{attribute 'TcRpcEnable' := '1'}
METHOD CheckState : HRESULT
VAR_INPUT
	hdl : UDINT; // Do not change, used by server.
END_VAR
VAR_OUTPUT
	bBusy : BOOL; // Do not change. Used by server to find out if the job is finished
	
	// List of OutputArguments for OPC UA method, may be customized
	State : BOOL; // Abgeschlossener MethodCall
	MethodCall: BOOL; //Input Recall
END_VAR
                        callCounterCheckState := callCounterCheckState + 1;
IF NOT jobFinished THEN
	bBusy := TRUE; // job is not finished yet
	CheckState := 0; // no error
ELSE
	bBusy := FALSE; // job is finished
	CheckState := 0; // done, no error occured during execution (OPC UA StatusCode "GOOD")
	jobFinished := FALSE;
	State := ResetCall;
	MethodCall := MethodCall_Name;
END_IF
                      
END_METHOD

{attribute 'TcRpcEnable' := '1'}
METHOD Start : HRESULT
VAR_INPUT
	// List of InputArguments for OPC UA method, may be customized
	MethodCall : BOOL; // some description
	DirectionPointA : BOOL;
	DirectionPointB : BOOL;
	EndschalterEntlastung : BOOL;	
END_VAR
VAR_OUTPUT
	hdl : UDINT; // Do not change, used by server.
END_VAR
                        callCounterStart := callCounterStart + 1;

MethodCall_Name := MethodCall;
DirectionPointA := Direction_01;
DirectionPointB := Direction_02;
EndschalterEntlastung := EndschalterEntlastung;

IF DirectionPointA := TRUE THEN
	DirectionPointB := FALSE;
END_IF

IF DirectionPointB := TRUE THEN
	DirectionPointA := FALSE;
END_IF

jobRunning := TRUE;
Start := 0; // no error occured, e.g. while parsing the input arguments (0 = OPC UA StatusCode "GOOD")
                      
END_METHOD
END_FUNCTION_BLOCK

FUNCTION_BLOCK HRL_OperatingModes
VAR_INPUT
	Start 			: BOOL;
	Stop			: BOOL;
	Reset			: BOOL;
	Schalter		: BOOL;
	Schrittkette_GS	: BOOL;
	Count1 : INT := 0;
	Count2 : INT := 0;
	Alt_abort: BOOL;
	Err_detected: BOOL;
	Diag_finished: BOOL;
	Alt_found: BOOL;
	Cycle_finished: BOOL;

END_VAR
VAR_OUTPUT
	{attribute 'OPC.UA.DA' := '1'} // für OPC UA freigeben
	A1 : BOOL := FALSE; //Initialzustand
	{attribute 'OPC.UA.DA' := '1'} // für OPC UA freigeben
	A2 : BOOL; //Stillstand angefordert am Ende des Zyklus
//	A3 : BOOL; //Stillstand angefordert in einem bestimmten Zustand
//	A4 : BOOL; //Erhaltener Stillstand
	{attribute 'OPC.UA.DA' := '1'} // für OPC UA freigeben
	A5 : BOOL; //Vorbereitung zur Wiederaufnahme nach Störung
	{attribute 'OPC.UA.DA' := '1'} // für OPC UA freigeben
	A6 : BOOL; //Fahrt in den Initialzustand
	{attribute 'OPC.UA.DA' := '1'} // für OPC UA freigeben
	F1 : BOOL; //Normalbetrieb
//	F2 : BOOL; //Anfahren
//	F3 : BOOL; //Abfahren
	{attribute 'OPC.UA.DA' := '1'} // für OPC UA freigeben
	F4 : BOOL; //Handbetrieb
//	F5 : BOOL; //Schrittbetrieb
//	F6 : BOOL; //Testbetrieb
	{attribute 'OPC.UA.DA' := '1'} // für OPC UA freigeben
	D1 : BOOL; //Not-Aus
	{attribute 'OPC.UA.DA' := '1'} // für OPC UA freigeben
	D2 : BOOL; //Diagnose und Störbehandlung
	{attribute 'OPC.UA.DA' := '1'} // für OPC UA freigeben
	D3 : BOOL; //Produktion trotz Störung
	MethodCall_InitStateDrive : BOOL;
	InputVar_InitStateDrive : BOOL;
END_VAR
VAR
	bFirstScan : BOOL := TRUE;
	FirstScanCount: INT := 0;
	AlwaysTrue : BOOL := TRUE;
	TestingVariable : BOOL;	
	 nTaskIdx : DINT;
	RS_InitialState: RS;
	RS_InitialState11: RS;	
	RS_InitialDrive: RS;
	RS_ManualOperationMode: RS;
	RS_AutomaticOperationMode: RS;
	RS_CycleEnded: RS;
	//Count: INT := 0;
	R_TRIG_Manual: R_TRIG;
	R_TRIG_Automatic: R_TRIG;
	R_TRIG_InitialDrive: R_TRIG;
	R_TRIG_CycleEnded: R_TRIG;
	R_TRIG_Init: R_TRIG;
	NeverTrue: BOOL := FALSE;
	SR_D1: SR;
	RS_D2: RS;
	
	RS_D3: RS;
	RS_A5: RS;
	
	
	bFirstCycle: BOOL;
END_VAR
  VAR  (* added by the conversion: wires and edge detectors of the diagram *)
    _EXECUTE50000000009_EN : BOOL;
  END_VAR

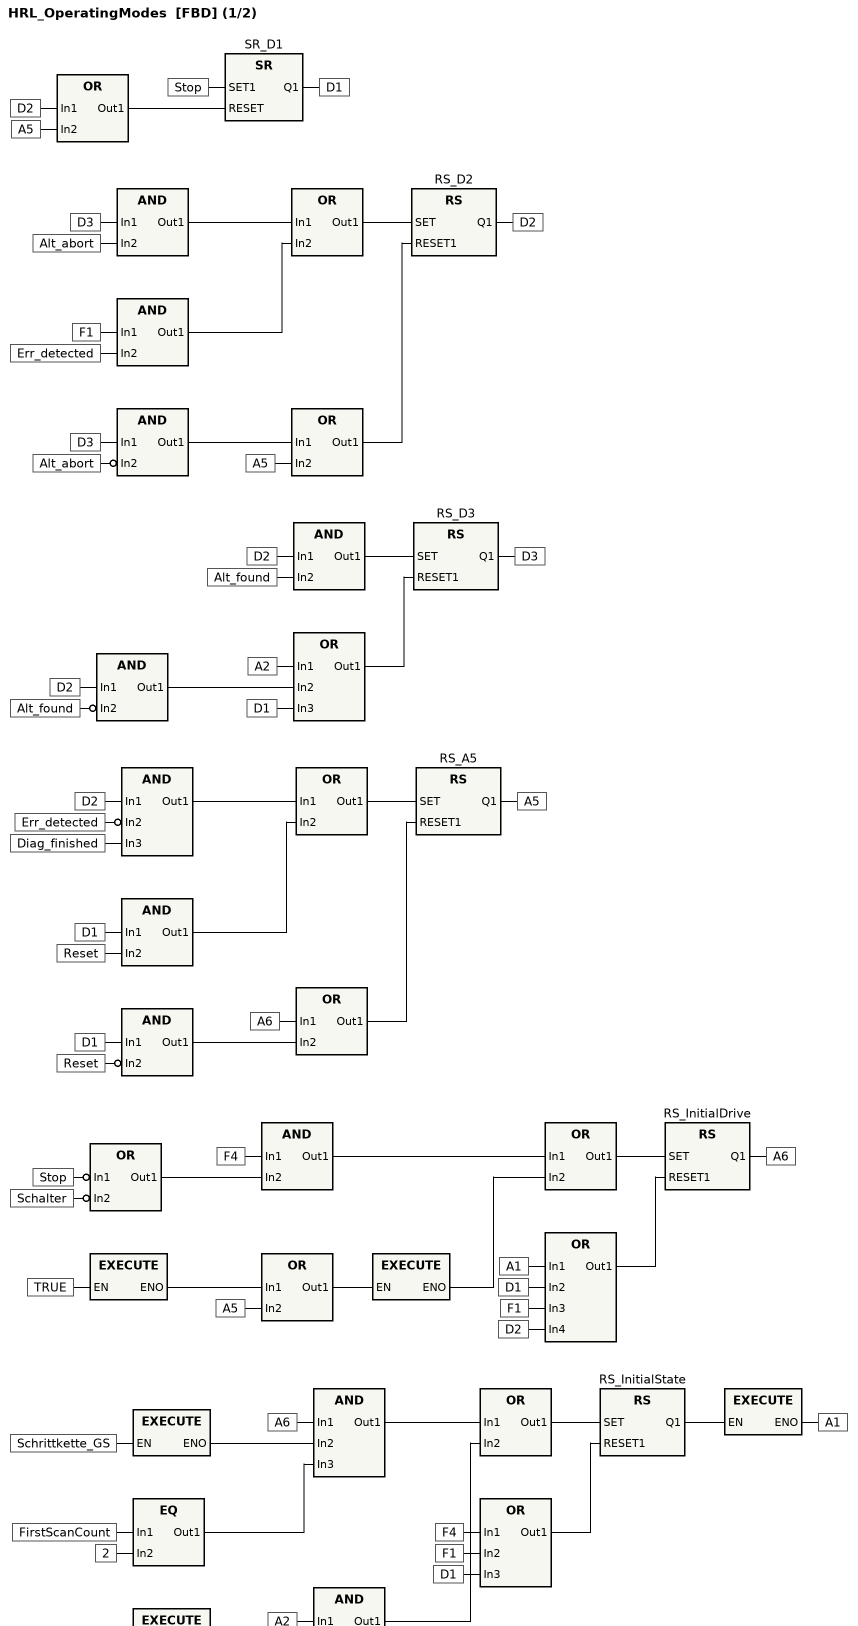
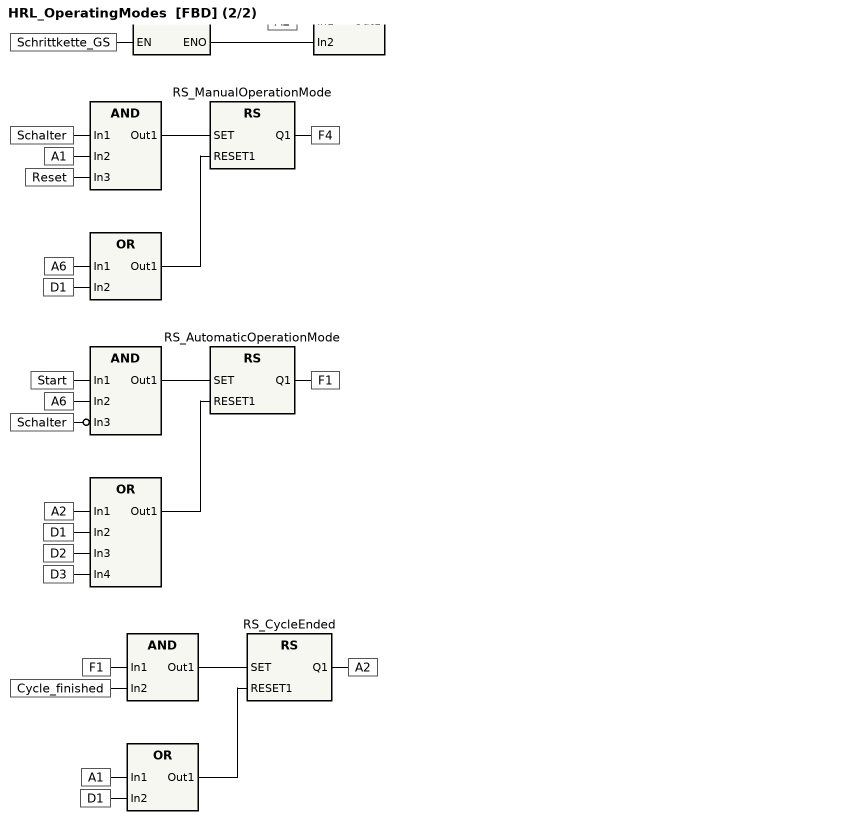
(* FBD diagram, written out as Structured Text *)
SR_D1(SET1 := Stop, RESET := D2 OR A5);
D1 := SR_D1.Q1;
RS_D2(SET := D3 AND Alt_abort OR F1 AND Err_detected, RESET1 := D3 AND NOT Alt_abort OR A5);
D2 := RS_D2.Q1;
RS_D3(SET := D2 AND Alt_found, RESET1 := A2 OR D2 AND NOT Alt_found OR D1);
D3 := RS_D3.Q1;
RS_A5(SET := D2 AND NOT Err_detected AND Diag_finished OR D1 AND Reset, RESET1 := A6 OR D1 AND NOT Reset);
A5 := RS_A5.Q1;
IF TRUE THEN
  nTaskIdx := GETCURTASKINDEXEX();
  
  IF nTaskIdx > 0 THEN
          bFirstCycle := _TaskInfo[nTaskIdx].FirstCycle;
  END_IF
END_IF;
_EXECUTE50000000009_EN := TRUE OR A5;
IF _EXECUTE50000000009_EN THEN
  IF AlwaysTrue THEN
      MethodCall_InitStateDrive := TRUE;
  	InputVar_InitStateDrive := TRUE;
  END_IF;
END_IF;
RS_InitialDrive(SET := F4 AND (NOT Stop OR NOT Schalter) OR _EXECUTE50000000009_EN, RESET1 := A1 OR D1 OR F1 OR D2);
A6 := RS_InitialDrive.Q1;
IF Schrittkette_GS THEN
  MethodCall_InitStateDrive := FALSE;
  InputVar_InitStateDrive := FALSE;
END_IF;
IF Schrittkette_GS THEN
  MethodCall_InitStateDrive := FALSE;
  InputVar_InitStateDrive := FALSE;
END_IF;
RS_InitialState(SET := A6 AND Schrittkette_GS AND FirstScanCount = 2 OR A2 AND Schrittkette_GS, RESET1 := F4 OR F1 OR D1);
IF RS_InitialState.Q1 THEN
  FirstScanCount := 0;
  bFirstScan := FALSE;
END_IF;
A1 := RS_InitialState.Q1;
RS_ManualOperationMode(SET := Schalter AND A1 AND Reset, RESET1 := A6 OR D1);
F4 := RS_ManualOperationMode.Q1;
RS_AutomaticOperationMode(SET := Start AND A6 AND NOT Schalter, RESET1 := A2 OR D1 OR D2 OR D3);
F1 := RS_AutomaticOperationMode.Q1;
RS_CycleEnded(SET := F1 AND Cycle_finished, RESET1 := A1 OR D1);
A2 := RS_CycleEnded.Q1;
END_FUNCTION_BLOCK

FUNCTION_BLOCK VSG_OperatingModes
VAR_INPUT
	Start 			: BOOL;
	Stop			: BOOL;
	Reset			: BOOL;
	Schalter		: BOOL;
	Schrittkette_GS	: BOOL;
	Count1 : INT := 0;
	Count2 : INT := 0;
	Alt_abort: BOOL;
	Err_detected: BOOL;
	Diag_finished: BOOL;
	Alt_found: BOOL;
	Cycle_finished: BOOL;

END_VAR
VAR_OUTPUT
	{attribute 'OPC.UA.DA' := '1'} // für OPC UA freigeben
	A1 : BOOL := FALSE; //Initialzustand
	{attribute 'OPC.UA.DA' := '1'} // für OPC UA freigeben
	A2 : BOOL; //Stillstand angefordert am Ende des Zyklus
//	A3 : BOOL; //Stillstand angefordert in einem bestimmten Zustand
//	A4 : BOOL; //Erhaltener Stillstand
	{attribute 'OPC.UA.DA' := '1'} // für OPC UA freigeben
	A5 : BOOL; //Vorbereitung zur Wiederaufnahme nach Störung
	{attribute 'OPC.UA.DA' := '1'} // für OPC UA freigeben
	A6 : BOOL; //Fahrt in den Initialzustand
	{attribute 'OPC.UA.DA' := '1'} // für OPC UA freigeben
	F1 : BOOL; //Normalbetrieb
//	F2 : BOOL; //Anfahren
//	F3 : BOOL; //Abfahren
	{attribute 'OPC.UA.DA' := '1'} // für OPC UA freigeben
	F4 : BOOL; //Handbetrieb
//	F5 : BOOL; //Schrittbetrieb
//	F6 : BOOL; //Testbetrieb
{attribute 'OPC.UA.DA' := '1'} // für OPC UA freigeben
	D1 : BOOL; //Not-Aus
	{attribute 'OPC.UA.DA' := '1'} // für OPC UA freigeben
	D2 : BOOL; //Diagnose und Störbehandlung
	{attribute 'OPC.UA.DA' := '1'} // für OPC UA freigeben
	D3 : BOOL; //Produktion trotz Störung
	MethodCall_InitStateDrive : BOOL;
	InputVar_InitStateDrive : BOOL;
END_VAR
VAR
	bFirstScan : BOOL := TRUE;
	FirstScanCount: INT := 0;
	AlwaysTrue : BOOL := TRUE;
	TestingVariable : BOOL;	
	 nTaskIdx : DINT;
	RS_InitialState: RS;
	RS_InitialState11: RS;	
	RS_InitialDrive: RS;
	RS_ManualOperationMode: RS;
	RS_AutomaticOperationMode: RS;
	RS_CycleEnded: RS;
	//Count: INT := 0;
	R_TRIG_Manual: R_TRIG;
	R_TRIG_Automatic: R_TRIG;
	R_TRIG_InitialDrive: R_TRIG;
	R_TRIG_CycleEnded: R_TRIG;
	R_TRIG_Init: R_TRIG;
	NeverTrue: BOOL := FALSE;
	SR_D1: SR;
	RS_D2: RS;
	
	RS_D3: RS;
	RS_A5: RS;
	
	
	bFirstCycle: BOOL;
END_VAR
  VAR  (* added by the conversion: wires and edge detectors of the diagram *)
    _EXECUTE50000000009_EN : BOOL;
  END_VAR

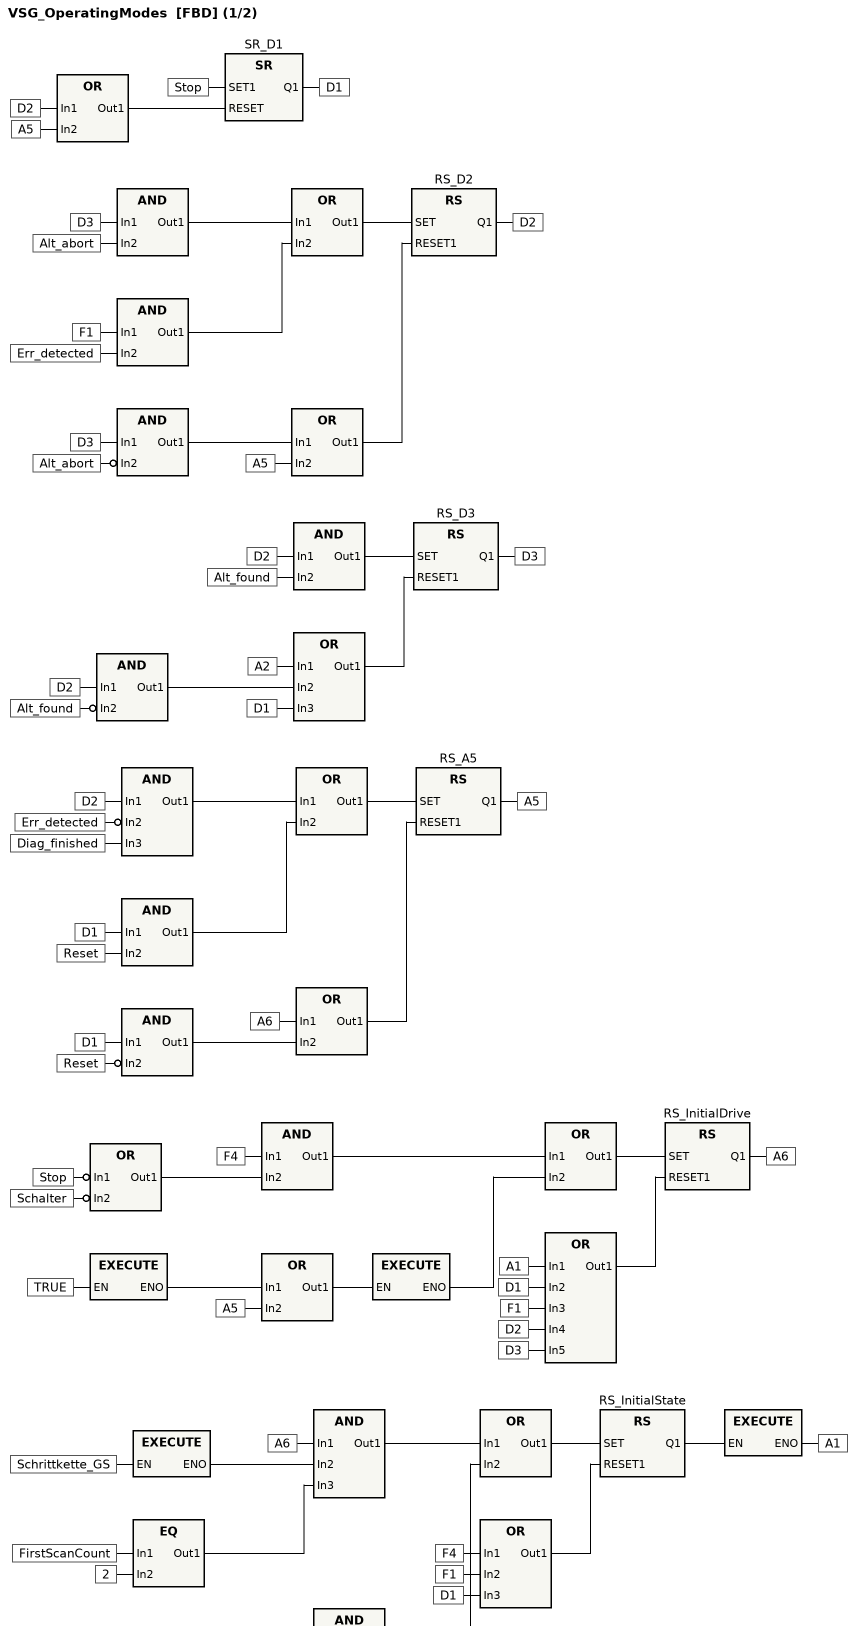
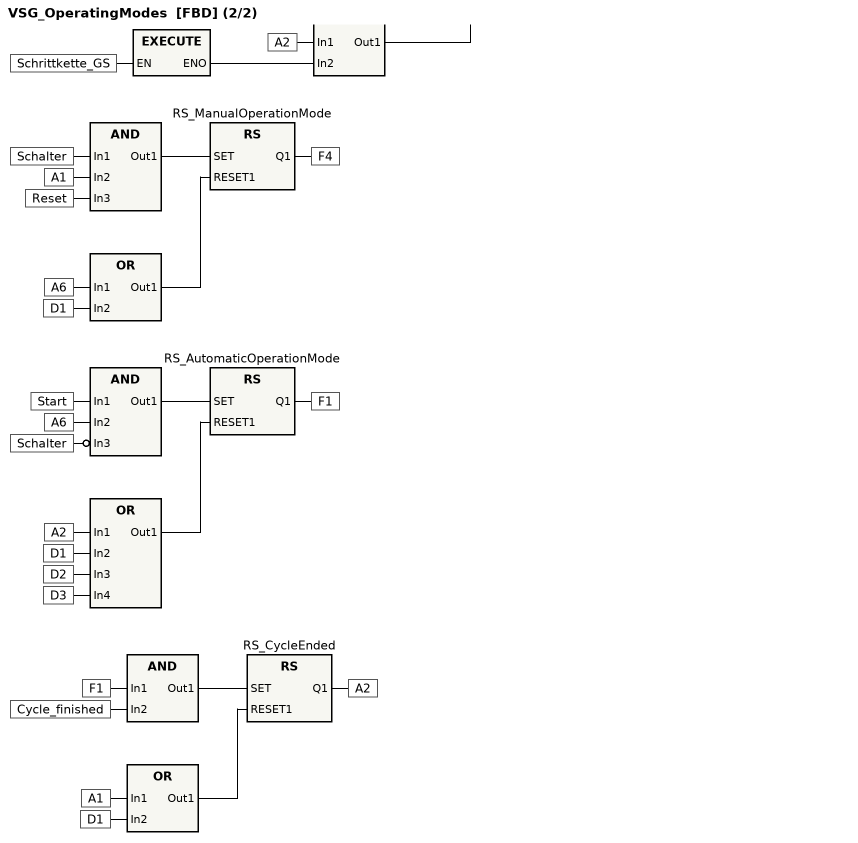
(* FBD diagram, written out as Structured Text *)
SR_D1(SET1 := Stop, RESET := D2 OR A5);
D1 := SR_D1.Q1;
RS_D2(SET := D3 AND Alt_abort OR F1 AND Err_detected, RESET1 := D3 AND NOT Alt_abort OR A5);
D2 := RS_D2.Q1;
RS_D3(SET := D2 AND Alt_found, RESET1 := A2 OR D2 AND NOT Alt_found OR D1);
D3 := RS_D3.Q1;
RS_A5(SET := D2 AND NOT Err_detected AND Diag_finished OR D1 AND Reset, RESET1 := A6 OR D1 AND NOT Reset);
A5 := RS_A5.Q1;
IF TRUE THEN
  nTaskIdx := GETCURTASKINDEXEX();
  
  IF nTaskIdx > 0 THEN
          bFirstCycle := _TaskInfo[nTaskIdx].FirstCycle;
  END_IF
END_IF;
_EXECUTE50000000009_EN := TRUE OR A5;
IF _EXECUTE50000000009_EN THEN
  IF AlwaysTrue THEN
      MethodCall_InitStateDrive := TRUE;
  	InputVar_InitStateDrive := TRUE;
  END_IF;
END_IF;
RS_InitialDrive(SET := F4 AND (NOT Stop OR NOT Schalter) OR _EXECUTE50000000009_EN, RESET1 := A1 OR D1 OR F1 OR D2 OR D3);
A6 := RS_InitialDrive.Q1;
IF Schrittkette_GS THEN
  MethodCall_InitStateDrive := FALSE;
  InputVar_InitStateDrive := FALSE;
END_IF;
IF Schrittkette_GS THEN
  MethodCall_InitStateDrive := FALSE;
  InputVar_InitStateDrive := FALSE;
END_IF;
RS_InitialState(SET := A6 AND Schrittkette_GS AND FirstScanCount = 2 OR A2 AND Schrittkette_GS, RESET1 := F4 OR F1 OR D1);
IF RS_InitialState.Q1 THEN
  FirstScanCount := 0;
  bFirstScan := FALSE;
END_IF;
A1 := RS_InitialState.Q1;
RS_ManualOperationMode(SET := Schalter AND A1 AND Reset, RESET1 := A6 OR D1);
F4 := RS_ManualOperationMode.Q1;
RS_AutomaticOperationMode(SET := Start AND A6 AND NOT Schalter, RESET1 := A2 OR D1 OR D2 OR D3);
F1 := RS_AutomaticOperationMode.Q1;
RS_CycleEnded(SET := F1 AND Cycle_finished, RESET1 := A1 OR D1);
A2 := RS_CycleEnded.Q1;
END_FUNCTION_BLOCK

FUNCTION_BLOCK MBS_OperatingModes
VAR_INPUT
	Start 			: BOOL;
	Stop			: BOOL;
	Reset			: BOOL;
	Schalter		: BOOL;
	Schrittkette_GS : BOOL;
END_VAR
VAR_OUTPUT
	A1 : BOOL; //Initialzustand
	A2 : BOOL; //Stillstand angefordert am Ende des Zyklus
//	A3 : BOOL; //Stillstand angefordert in einem bestimmten Zustand
//	A4 : BOOL; //Erhaltener Stillstand
//	A5 : BOOL; //Vorbereitung zur Wiederaufnahme nach Störung
	A6 : BOOL; //Fahrt in den Initialzustand
	F1 : BOOL; //Normalbetrieb
//	F2 : BOOL; //Anfahren
//	F3 : BOOL; //Abfahren
	F4 : BOOL; //Handbetrieb
//	F5 : BOOL; //Schrittbetrieb
//	F6 : BOOL; //Testbetrieb
//	D1 : BOOL; //Not-Aus
//	D2 : BOOL; //DIagnose und Störbehandlung
//	D3 : BOOL; //Produktion trotz Störung
END_VAR
VAR
	bFirstScan : BOOL := TRUE;	
	
	RS_InitialState: RS;	
	RS_InitialDrive: RS;
	RS_ManualOperationMode: RS;
	RS_AutomaticOperationMode: RS;
	RS_CycleEnded: RS;

	R_TRIG_Manual: R_TRIG;
	R_TRIG_Automatic: R_TRIG;
	R_TRIG_InitialDrive: R_TRIG;
	R_TRIG_CycleEnded: R_TRIG;
	R_TRIG_Init: R_TRIG;
END_VAR

                  R_TRIG_InitialDrive(CLK := RS_InitialDrive);
R_TRIG_CycleEnded(CLK := RS_CycleEnded);
R_TRIG_Manual(CLK := RS_ManualOperationMode);
R_TRIG_Automatic(CLK := RS_AutomaticOperationMode);
RS_InitialState(SET := ((((R_TRIG_InitialDrive.Q) AND (Schrittkette_GS))) OR (((R_TRIG_CycleEnded.Q) AND (Schrittkette_GS)))), RESET1 := ((R_TRIG_Manual.Q) OR (R_TRIG_Automatic.Q)));
A1 := RS_InitialState.Q1;
RS_ManualOperationMode(SET := ((Schalter) AND (A1) AND (Reset)), RESET1 := A6);
F4 := RS_ManualOperationMode.Q1;
R_TRIG_Manual(CLK := RS_ManualOperationMode);
R_TRIG_Init(CLK := RS_InitialState);
RS_InitialDrive(SET := ((((R_TRIG_Manual.Q) AND (((Stop) OR (NOT (Schalter)))))) OR ((bFirstScan))), RESET1 := R_TRIG_Init.Q);
A6 := RS_InitialDrive.Q1;
R_TRIG_Init(CLK := RS_InitialState);
R_TRIG_CycleEnded(CLK := RS_CycleEnded);
RS_AutomaticOperationMode(SET := ((Start) AND (R_TRIG_Init.Q) AND (NOT (Schalter))), RESET1 := R_TRIG_CycleEnded.Q);
F1 := RS_AutomaticOperationMode.Q1;
R_TRIG_Automatic(CLK := RS_AutomaticOperationMode);
R_TRIG_Init(CLK := RS_InitialState);
RS_CycleEnded(SET := ((R_TRIG_Automatic.Q) AND (((Schalter) OR (Stop)))), RESET1 := R_TRIG_Init.Q);
A2 := RS_CycleEnded.Q1;
                
END_FUNCTION_BLOCK

FUNCTION_BLOCK SST_OperatingModes
VAR_INPUT
	Start 			: BOOL;
	Stop			: BOOL;
	Reset			: BOOL;
	Schalter		: BOOL;
	Schrittkette_GS : BOOL;
END_VAR
VAR_OUTPUT
	A1 : BOOL; //Initialzustand
	A2 : BOOL; //Stillstand angefordert am Ende des Zyklus
//	A3 : BOOL; //Stillstand angefordert in einem bestimmten Zustand
//	A4 : BOOL; //Erhaltener Stillstand
//	A5 : BOOL; //Vorbereitung zur Wiederaufnahme nach Störung
	A6 : BOOL; //Fahrt in den Initialzustand
	F1 : BOOL; //Normalbetrieb
//	F2 : BOOL; //Anfahren
//	F3 : BOOL; //Abfahren
	F4 : BOOL; //Handbetrieb
//	F5 : BOOL; //Schrittbetrieb
//	F6 : BOOL; //Testbetrieb
//	D1 : BOOL; //Not-Aus
//	D2 : BOOL; //DIagnose und Störbehandlung
//	D3 : BOOL; //Produktion trotz Störung
END_VAR
VAR
	bFirstScan : BOOL := TRUE;	
	
	RS_InitialState: RS;	
	RS_InitialDrive: RS;
	RS_ManualOperationMode: RS;
	RS_AutomaticOperationMode: RS;
	RS_CycleEnded: RS;

	R_TRIG_Manual: R_TRIG;
	R_TRIG_Automatic: R_TRIG;
	R_TRIG_InitialDrive: R_TRIG;
	R_TRIG_CycleEnded: R_TRIG;
	R_TRIG_Init: R_TRIG;
END_VAR

                  R_TRIG_InitialDrive(CLK := RS_InitialDrive);
R_TRIG_CycleEnded(CLK := RS_CycleEnded);
R_TRIG_Manual(CLK := RS_ManualOperationMode);
R_TRIG_Automatic(CLK := RS_AutomaticOperationMode);
RS_InitialState(SET := ((((R_TRIG_InitialDrive.Q) AND (Schrittkette_GS))) OR (((R_TRIG_CycleEnded.Q) AND (Schrittkette_GS)))), RESET1 := ((R_TRIG_Manual.Q) OR (R_TRIG_Automatic.Q)));
A1 := RS_InitialState.Q1;
RS_ManualOperationMode(SET := ((Schalter) AND (A1) AND (Reset)), RESET1 := A6);
F4 := RS_ManualOperationMode.Q1;
R_TRIG_Manual(CLK := RS_ManualOperationMode);
R_TRIG_Init(CLK := RS_InitialState);
RS_InitialDrive(SET := ((((R_TRIG_Manual.Q) AND (((Stop) OR (NOT (Schalter)))))) OR ((bFirstScan))), RESET1 := R_TRIG_Init.Q);
A6 := RS_InitialDrive.Q1;
R_TRIG_Init(CLK := RS_InitialState);
R_TRIG_CycleEnded(CLK := RS_CycleEnded);
RS_AutomaticOperationMode(SET := ((Start) AND (R_TRIG_Init.Q) AND (NOT (Schalter))), RESET1 := R_TRIG_CycleEnded.Q);
F1 := RS_AutomaticOperationMode.Q1;
R_TRIG_Automatic(CLK := RS_AutomaticOperationMode);
R_TRIG_Init(CLK := RS_InitialState);
RS_CycleEnded(SET := ((R_TRIG_Automatic.Q) AND (((Schalter) OR (Stop)))), RESET1 := R_TRIG_Init.Q);
A2 := RS_CycleEnded.Q1;

                
END_FUNCTION_BLOCK

FUNCTION_BLOCK VSG_OperatingModes_alt
VAR_INPUT
	Start 			: BOOL;
	Stop			: BOOL;
	Reset			: BOOL;
	Schalter		: BOOL;
	Schrittkette_GS : BOOL;
END_VAR
VAR_OUTPUT
	A1 : BOOL; //Initialzustand
	A2 : BOOL; //Stillstand angefordert am Ende des Zyklus
//	A3 : BOOL; //Stillstand angefordert in einem bestimmten Zustand
//	A4 : BOOL; //Erhaltener Stillstand
//	A5 : BOOL; //Vorbereitung zur Wiederaufnahme nach Störung
	A6 : BOOL; //Fahrt in den Initialzustand
	F1 : BOOL; //Normalbetrieb
//	F2 : BOOL; //Anfahren
//	F3 : BOOL; //Abfahren
	F4 : BOOL; //Handbetrieb
//	F5 : BOOL; //Schrittbetrieb
//	F6 : BOOL; //Testbetrieb
//	D1 : BOOL; //Not-Aus
//	D2 : BOOL; //DIagnose und Störbehandlung
//	D3 : BOOL; //Produktion trotz Störung
END_VAR
VAR
	bFirstScan : BOOL := TRUE;	
	
	RS_InitialState: RS;	
	RS_InitialDrive: RS;
	RS_ManualOperationMode: RS;
	RS_AutomaticOperationMode: RS;
	RS_CycleEnded: RS;

	R_TRIG_Manual: R_TRIG;
	R_TRIG_Automatic: R_TRIG;
	R_TRIG_InitialDrive: R_TRIG;
	R_TRIG_CycleEnded: R_TRIG;
	R_TRIG_Init: R_TRIG;
END_VAR

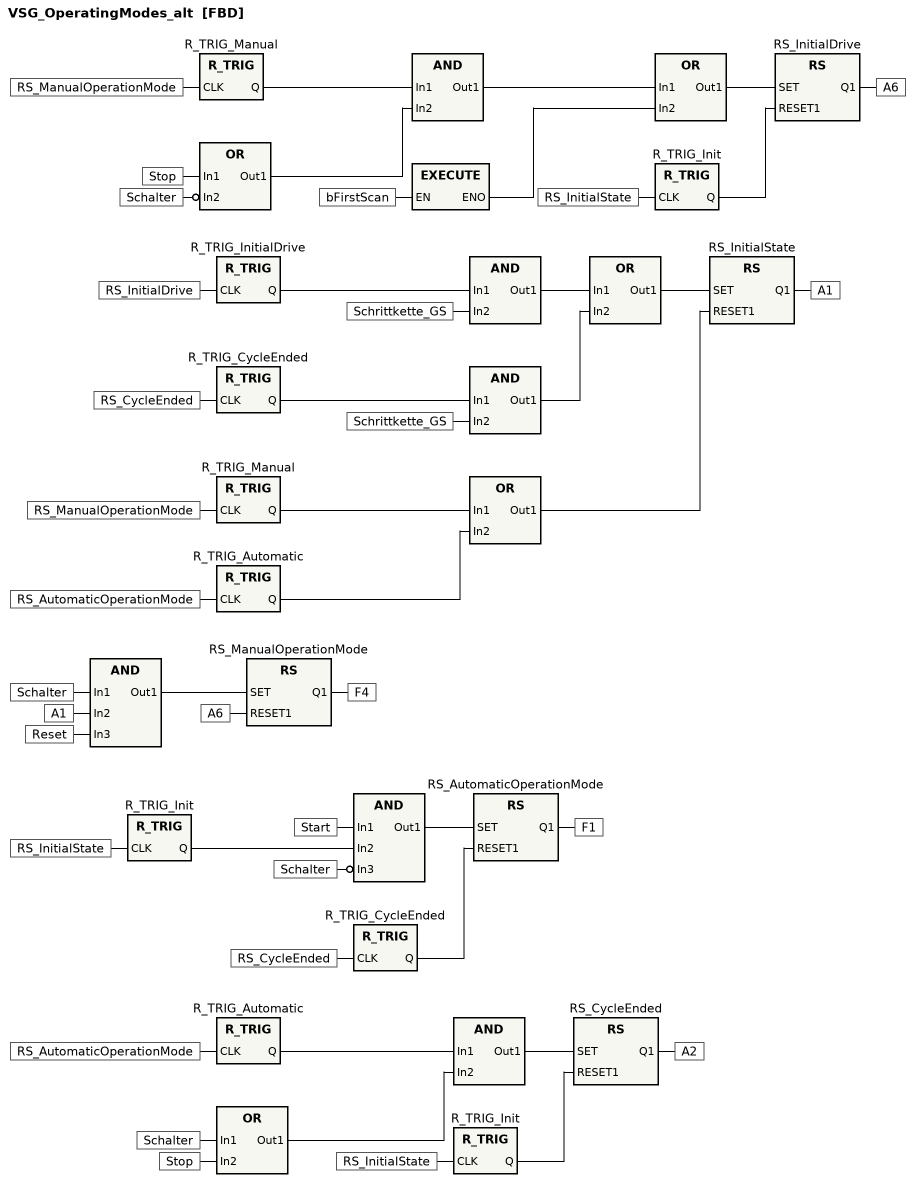
(* FBD diagram, written out as Structured Text *)
R_TRIG_Manual(CLK := RS_ManualOperationMode);
IF bFirstScan THEN
  IF bFirstScan THEN
      // Code, der nur beim ersten Scan ausgeführt werden soll
      // Zum Beispiel: Initialisierung von Parametern, Setzen von Startwerten etc.
  	VSG_SkillSet.MethodCall_InitStateDrive := TRUE;
  	VSG_SkillSet.InputVar_InitStateDrive := TRUE;
      bFirstScan := FALSE; // Nach der Ausführung die Variable zurücksetzen
  END_IF;
END_IF;
R_TRIG_Init(CLK := RS_InitialState);
RS_InitialDrive(SET := R_TRIG_Manual.Q AND (Stop OR NOT Schalter) OR bFirstScan, RESET1 := R_TRIG_Init.Q);
A6 := RS_InitialDrive.Q1;
R_TRIG_InitialDrive(CLK := RS_InitialDrive);
R_TRIG_CycleEnded(CLK := RS_CycleEnded);
R_TRIG_Manual(CLK := RS_ManualOperationMode);
R_TRIG_Automatic(CLK := RS_AutomaticOperationMode);
RS_InitialState(SET := R_TRIG_InitialDrive.Q AND Schrittkette_GS OR R_TRIG_CycleEnded.Q AND Schrittkette_GS, RESET1 := R_TRIG_Manual.Q OR R_TRIG_Automatic.Q);
A1 := RS_InitialState.Q1;
RS_ManualOperationMode(SET := Schalter AND A1 AND Reset, RESET1 := A6);
F4 := RS_ManualOperationMode.Q1;
R_TRIG_Init(CLK := RS_InitialState);
R_TRIG_CycleEnded(CLK := RS_CycleEnded);
RS_AutomaticOperationMode(SET := Start AND R_TRIG_Init.Q AND NOT Schalter, RESET1 := R_TRIG_CycleEnded.Q);
F1 := RS_AutomaticOperationMode.Q1;
R_TRIG_Automatic(CLK := RS_AutomaticOperationMode);
R_TRIG_Init(CLK := RS_InitialState);
RS_CycleEnded(SET := R_TRIG_Automatic.Q AND (Schalter OR Stop), RESET1 := R_TRIG_Init.Q);
A2 := RS_CycleEnded.Q1;
END_FUNCTION_BLOCK

{attribute 'OPC.UA.DA.JobMethod' := 'JobMethode_HorizontalMove'}
FUNCTION_BLOCK HRL_CB_AS_HorizontalMoveSensors
VAR
	AlwaysTrue : BOOL := TRUE;
	// Used for debugging purposes to display InputArguments of method call
	MethodCall_HorizontalMove : BOOL := FALSE; // used to store InputArg "MethodCall" from Start() method
	ResetMethodCall	: BOOL := FALSE;
	DirectionHorizontal : BOOL; // defines movement direction
	callCounterStart : ULINT; // counts how many times the Start() method has been called
	callCounterCheckState : ULINT; // counts how many times the CheckState() method has been called
	callCounterAbort : ULINT; // counts how many times the Abort() method has been called
	
	// Variables to determine if a job has been started (Start() method has been called) or finished
	jobRunning : BOOL;
	jobFinished : BOOL;

	// State machine variable
	state : UDINT;
	
	// FB Intatziation Variable
	HRL_CB_HorizontalMove : AxisControl_MultipleInputSensors;
END_VAR
	
VAR_INPUT
	ESS						: BOOL;
	LightBarrierSensor_01 	: BOOL;
	LightBarrierSensor_02 	: BOOL;
	AutomaticMode			: BOOL;
END_VAR

VAR_OUTPUT
	DO_MovingConveyorBelt : BOOL;
END_VAR

                  HRL_CB_HorizontalMove(
    MethodCall := MethodCall_HorizontalMove,
    EmergencyStopSignal := ESS,
    Direction := DirectionHorizontal,
    InitStateDrive_Input := FALSE,
    DI01 := LightBarrierSensor_01,
    DI02 := LightBarrierSensor_02,
    TouchSensorRelief := FALSE,
    TOF_Time_MotorControl := T#0MS,
    TOF_Time_TouchSensorRelief := T#0MS,
    OperatingMode := AutomaticMode
);
DO_MovingConveyorBelt := HRL_CB_HorizontalMove.DigitalOutputControl_01;

                

{attribute 'TcRpcEnable' := '1'}
METHOD Abort : HRESULT
VAR_INPUT
	hdl : UDINT; // Do not change, used by server.
END_VAR
                        callCounterAbort := callCounterAbort + 1;

                      
END_METHOD

{attribute 'TcRpcEnable' := '1'}
METHOD CheckState : HRESULT
VAR_INPUT
	hdl : UDINT; // Do not change, used by server.
END_VAR
VAR_OUTPUT
	bBusy : BOOL; // Do not change. Used by server to find out if the job is finished
	
	// List of OutputArguments for OPC UA method, may be customized
	State : BOOL; // Abgeschlossener MethodCall
	MethodCall: BOOL; //Input Recall
END_VAR
                        callCounterCheckState := callCounterCheckState + 1;
IF NOT jobFinished THEN
	bBusy := TRUE; // job is not finished yet
	CheckState := 0; // no error
ELSE
	bBusy := FALSE; // job is finished
	CheckState := 0; // done, no error occured during execution (OPC UA StatusCode "GOOD")
	jobFinished := FALSE;
	State := ResetMethodCall;
	MethodCall := MethodCall_HorizontalMove;
END_IF
                      
END_METHOD

{attribute 'TcRpcEnable' := '1'}
METHOD Start : HRESULT
VAR_INPUT
	// List of InputArguments for OPC UA method, may be customized
	MethodCall : BOOL; // some description
	MovementDirection : BOOL;	
END_VAR
VAR_OUTPUT
	hdl : UDINT; // Do not change, used by server.
END_VAR
                        callCounterStart := callCounterStart + 1;

MethodCall_HorizontalMove := MethodCall;
DirectionHorizontal := MovementDirection;

jobRunning := TRUE;
Start := 0; // no error occured, e.g. while parsing the input arguments (0 = OPC UA StatusCode "GOOD")
                      
END_METHOD
END_FUNCTION_BLOCK

{attribute 'OPC.UA.DA.JobMethod' := 'HRL_NMethod_Auslagern'}
FUNCTION_BLOCK HRL_NMethod_Auslagern
VAR_INPUT
    ESS_OK : BOOL;
    AutomaticMode : BOOL;

    HRL_Enc_horizontal_I1 : UDINT;
    HRL_Enc_horizontal_I2 : UDINT;
    HRL_Enc_vertikal_I1 : UDINT;
    HRL_Enc_vertikal_I2 : UDINT;

    HRL_Ref_Taster_horizontal : BOOL;
    HRL_Ref_Taster_vertikal : BOOL;
    HRL_Ref_Taster_Ausleger_vorne : BOOL;
    HRL_Ref_Taster_Ausleger_hinten : BOOL;

    HRL_LS_innen : BOOL;
    HRL_LS_aussen : BOOL;
END_VAR

VAR_OUTPUT
    REQ_CB_forwards : BOOL;
    REQ_CB_backwards : BOOL;

    REQ_RGB_Forwards : BOOL;
    REQ_RGB_Backwards : BOOL;

    REQ_RGB_VerticalDown : BOOL;
    REQ_RGB_VerticalUp : BOOL;

    REQ_RGB_HorizontalForward : BOOL;
    REQ_RGB_HorizontalBackward : BOOL;

    Busy : BOOL;
    Done : BOOL;
    Error : BOOL;
    ErrorId : UDINT;
    CurrentStep : UDINT;
END_VAR

VAR
    MethodCall_Auslagern : BOOL := FALSE;

    callCounterStart : ULINT := 0;
    callCounterAbort : ULINT := 0;
    callCounterCheckState : ULINT := 0;

    jobRunning : BOOL := FALSE;
    jobFinished : BOOL := FALSE;

    step : UDINT := 0;
    lastStep : UDINT := 0;
    bStepChanged : BOOL := FALSE;

    TargetHorizontalShelf_I1 : UDINT := 0;
    TargetHorizontalShelf_I2 : UDINT := 0;
    TargetVerticalShelf_I1 : UDINT := 0;
    TargetVerticalShelf_I2 : UDINT := 0;

    TargetHorizontalTransfer_I1 : UDINT := 0;
    TargetHorizontalTransfer_I2 : UDINT := 0;
    TargetVerticalTransfer_I1 : UDINT := 0;
    TargetVerticalTransfer_I2 : UDINT := 0;

    ActiveTargetHorizontal_I1 : UDINT := 0;
    ActiveTargetHorizontal_I2 : UDINT := 0;
    ActiveTargetVertical_I1 : UDINT := 0;
    ActiveTargetVertical_I2 : UDINT := 0;

    WatchdogTime : TIME := T#15S;

    cmdHorizontal : BOOL := FALSE;
    cmdVertical : BOOL := FALSE;
    cmdAuslegerForward : BOOL := FALSE;
    cmdAuslegerBackward : BOOL := FALSE;
    cmdConveyorForward : BOOL := FALSE;

    dirHorizontalToRegal : BOOL := FALSE;
    dirVerticalDown : BOOL := FALSE;

    bOppositeCommandError : BOOL := FALSE;
    bAbortRequest : BOOL := FALSE;

    fbHorizontal : AxisControl_Encoder;
    fbVertical : AxisControl_Encoder;
    fbAuslegerForward : AxisControl_MultipleInputSensors;
    fbAuslegerBackward : AxisControl_MultipleInputSensors;
    fbConveyorForward : AxisControl_MultipleInputSensors;

    tonWatchdog : TON;
END_VAR

                  REQ_CB_forwards := FALSE;
REQ_CB_backwards := FALSE;

REQ_RGB_Forwards := FALSE;
REQ_RGB_Backwards := FALSE;

REQ_RGB_VerticalDown := FALSE;
REQ_RGB_VerticalUp := FALSE;

REQ_RGB_HorizontalForward := FALSE;
REQ_RGB_HorizontalBackward := FALSE;

bOppositeCommandError := FALSE;

bStepChanged := (step <> lastStep);
lastStep := step;

IF bAbortRequest THEN
    cmdHorizontal := FALSE;
    cmdVertical := FALSE;
    cmdAuslegerForward := FALSE;
    cmdAuslegerBackward := FALSE;
    cmdConveyorForward := FALSE;

    MethodCall_Auslagern := FALSE;

    Busy := FALSE;
    Done := FALSE;

    jobRunning := FALSE;
    jobFinished := TRUE;

    // Fehlerstatus bewusst nicht überschreiben
    step := 0;
    bAbortRequest := FALSE;
END_IF;

IF bStepChanged THEN
    tonWatchdog(IN := FALSE, PT := WatchdogTime);
END_IF;

tonWatchdog(
    IN := jobRunning AND (step <> 0) AND (step <> 100) AND (step <> 900),
    PT := WatchdogTime
);

IF tonWatchdog.Q THEN
    Error := TRUE;
    ErrorId := 100;
    step := 900;
END_IF;

IF jobRunning AND NOT ESS_OK THEN
    Error := TRUE;
    ErrorId := 1;
    step := 900;
END_IF;

IF jobRunning AND NOT AutomaticMode THEN
    Error := TRUE;
    ErrorId := 2;
    step := 900;
END_IF;

IF step = 50 THEN
    ActiveTargetHorizontal_I1 := TargetHorizontalTransfer_I1;
    ActiveTargetHorizontal_I2 := TargetHorizontalTransfer_I2;
ELSE
    ActiveTargetHorizontal_I1 := TargetHorizontalShelf_I1;
    ActiveTargetHorizontal_I2 := TargetHorizontalShelf_I2;
END_IF;

IF step = 60 THEN
    ActiveTargetVertical_I1 := TargetVerticalTransfer_I1;
    ActiveTargetVertical_I2 := TargetVerticalTransfer_I2;
ELSE
    ActiveTargetVertical_I1 := TargetVerticalShelf_I1;
    ActiveTargetVertical_I2 := TargetVerticalShelf_I2;
END_IF;

dirHorizontalToRegal := (HRL_Enc_horizontal_I1 < ActiveTargetHorizontal_I1);
dirVerticalDown := (HRL_Enc_vertikal_I1 < ActiveTargetVertical_I1);

fbHorizontal(
    MethodCall := cmdHorizontal,
    EmergencyStopSignal := NOT ESS_OK,
    Direction := dirHorizontalToRegal,
    InitStateDrive_Input := FALSE,
    DI01 := HRL_Ref_Taster_horizontal,
    DI02_EncoderStart01 := HRL_Enc_horizontal_I1,
    DI03_EncoderTarget01 := ActiveTargetHorizontal_I1,
    DI04_EncoderStart02 := HRL_Enc_horizontal_I2,
    DI05_EncoderTarget02 := ActiveTargetHorizontal_I2,
    TouchSensorRelief := FALSE,
    TOF_Time_MotorControl := T#0MS,
    TOF_Time_TouchSensorRelief := T#0MS,
    OperatingMode := AutomaticMode
);

fbVertical(
    MethodCall := cmdVertical,
    EmergencyStopSignal := NOT ESS_OK,
    Direction := dirVerticalDown,
    InitStateDrive_Input := FALSE,
    DI01 := HRL_Ref_Taster_vertikal,
    DI02_EncoderStart01 := HRL_Enc_vertikal_I1,
    DI03_EncoderTarget01 := ActiveTargetVertical_I1,
    DI04_EncoderStart02 := HRL_Enc_vertikal_I2,
    DI05_EncoderTarget02 := ActiveTargetVertical_I2,
    TouchSensorRelief := FALSE,
    TOF_Time_MotorControl := T#0MS,
    TOF_Time_TouchSensorRelief := T#0MS,
    OperatingMode := AutomaticMode
);

fbAuslegerForward(
    MethodCall := cmdAuslegerForward,
    EmergencyStopSignal := NOT ESS_OK,
    Direction := TRUE,
    InitStateDrive_Input := FALSE,
    DI01 := HRL_Ref_Taster_Ausleger_hinten,
    DI02 := HRL_Ref_Taster_Ausleger_vorne,
    TouchSensorRelief := FALSE,
    TOF_Time_MotorControl := T#0MS,
    TOF_Time_TouchSensorRelief := T#0MS,
    OperatingMode := AutomaticMode
);

fbAuslegerBackward(
    MethodCall := cmdAuslegerBackward,
    EmergencyStopSignal := NOT ESS_OK,
    Direction := TRUE,
    InitStateDrive_Input := FALSE,
    DI01 := HRL_Ref_Taster_Ausleger_vorne,
    DI02 := HRL_Ref_Taster_Ausleger_hinten,
    TouchSensorRelief := FALSE,
    TOF_Time_MotorControl := T#0MS,
    TOF_Time_TouchSensorRelief := T#0MS,
    OperatingMode := AutomaticMode
);

fbConveyorForward(
    MethodCall := cmdConveyorForward,
    EmergencyStopSignal := NOT ESS_OK,
    Direction := TRUE,
    InitStateDrive_Input := FALSE,
    DI01 := HRL_LS_innen,
    DI02 := HRL_LS_aussen,
    TouchSensorRelief := FALSE,
    TOF_Time_MotorControl := T#0MS,
    TOF_Time_TouchSensorRelief := T#0MS,
    OperatingMode := AutomaticMode
);

CASE step OF

    0:
        Busy := FALSE;

        cmdHorizontal := FALSE;
        cmdVertical := FALSE;
        cmdAuslegerForward := FALSE;
        cmdAuslegerBackward := FALSE;
        cmdConveyorForward := FALSE;

        jobRunning := FALSE;

        // WICHTIG:
        // Done, Error, ErrorId und jobFinished hier NICHT pauschal löschen.
        // Diese Werte bleiben stehen, bis ein neuer Auftrag startet.

        IF MethodCall_Auslagern THEN

            IF NOT ESS_OK THEN
                Error := TRUE;
                ErrorId := 1;
                MethodCall_Auslagern := FALSE;
                jobFinished := TRUE;
                step := 900;

            ELSIF NOT AutomaticMode THEN
                Error := TRUE;
                ErrorId := 2;
                MethodCall_Auslagern := FALSE;
                jobFinished := TRUE;
                step := 900;

            ELSE
                Done := FALSE;
                Error := FALSE;
                ErrorId := 0;

                Busy := TRUE;
                jobRunning := TRUE;
                jobFinished := FALSE;

                step := 10;
            END_IF;

        END_IF;


    10:
        Busy := TRUE;

        cmdHorizontal := TRUE;
        cmdVertical := FALSE;
        cmdAuslegerForward := FALSE;
        cmdAuslegerBackward := FALSE;
        cmdConveyorForward := FALSE;

        IF dirHorizontalToRegal THEN
            REQ_RGB_HorizontalForward := fbHorizontal.DigitalOutputControl_01;
        ELSE
            REQ_RGB_HorizontalBackward := fbHorizontal.DigitalOutputControl_01;
        END_IF;

        IF REQ_RGB_HorizontalForward AND REQ_RGB_HorizontalBackward THEN
            Error := TRUE;
            ErrorId := 200;
            step := 900;
        END_IF;

        IF fbHorizontal.ResetMethodCall THEN
            cmdHorizontal := FALSE;
            step := 20;
        END_IF;


    20:
        Busy := TRUE;

        cmdHorizontal := FALSE;
        cmdVertical := TRUE;
        cmdAuslegerForward := FALSE;
        cmdAuslegerBackward := FALSE;
        cmdConveyorForward := FALSE;

        IF dirVerticalDown THEN
            REQ_RGB_VerticalDown := fbVertical.DigitalOutputControl_01;
        ELSE
            REQ_RGB_VerticalUp := fbVertical.DigitalOutputControl_01;
        END_IF;

        IF REQ_RGB_VerticalDown AND REQ_RGB_VerticalUp THEN
            Error := TRUE;
            ErrorId := 201;
            step := 900;
        END_IF;

        IF fbVertical.ResetMethodCall THEN
            cmdVertical := FALSE;
            step := 30;
        END_IF;


    30:
        Busy := TRUE;

        cmdHorizontal := FALSE;
        cmdVertical := FALSE;
        cmdAuslegerForward := TRUE;
        cmdAuslegerBackward := FALSE;
        cmdConveyorForward := FALSE;

        REQ_RGB_Forwards := fbAuslegerForward.DigitalOutputControl_01;

        IF REQ_RGB_Forwards AND REQ_RGB_Backwards THEN
            Error := TRUE;
            ErrorId := 202;
            step := 900;
        END_IF;

        IF fbAuslegerForward.ResetMethodCall THEN
            cmdAuslegerForward := FALSE;
            step := 40;
        END_IF;


    40:
        Busy := TRUE;

        cmdHorizontal := FALSE;
        cmdVertical := FALSE;
        cmdAuslegerForward := FALSE;
        cmdAuslegerBackward := TRUE;
        cmdConveyorForward := FALSE;

        REQ_RGB_Backwards := fbAuslegerBackward.DigitalOutputControl_01;

        IF REQ_RGB_Forwards AND REQ_RGB_Backwards THEN
            Error := TRUE;
            ErrorId := 203;
            step := 900;
        END_IF;

        IF fbAuslegerBackward.ResetMethodCall THEN
            cmdAuslegerBackward := FALSE;
            step := 50;
        END_IF;


    50:
        Busy := TRUE;

        cmdHorizontal := TRUE;
        cmdVertical := FALSE;
        cmdAuslegerForward := FALSE;
        cmdAuslegerBackward := FALSE;
        cmdConveyorForward := FALSE;

        IF dirHorizontalToRegal THEN
            REQ_RGB_HorizontalForward := fbHorizontal.DigitalOutputControl_01;
        ELSE
            REQ_RGB_HorizontalBackward := fbHorizontal.DigitalOutputControl_01;
        END_IF;

        IF REQ_RGB_HorizontalForward AND REQ_RGB_HorizontalBackward THEN
            Error := TRUE;
            ErrorId := 204;
            step := 900;
        END_IF;

        IF fbHorizontal.ResetMethodCall THEN
            cmdHorizontal := FALSE;
            step := 60;
        END_IF;


    60:
        Busy := TRUE;

        cmdHorizontal := FALSE;
        cmdVertical := TRUE;
        cmdAuslegerForward := FALSE;
        cmdAuslegerBackward := FALSE;
        cmdConveyorForward := FALSE;

        IF dirVerticalDown THEN
            REQ_RGB_VerticalDown := fbVertical.DigitalOutputControl_01;
        ELSE
            REQ_RGB_VerticalUp := fbVertical.DigitalOutputControl_01;
        END_IF;

        IF REQ_RGB_VerticalDown AND REQ_RGB_VerticalUp THEN
            Error := TRUE;
            ErrorId := 205;
            step := 900;
        END_IF;

        IF fbVertical.ResetMethodCall THEN
            cmdVertical := FALSE;
            step := 65;
        END_IF;


    65:
        Busy := TRUE;

        cmdHorizontal := FALSE;
        cmdVertical := FALSE;
        cmdAuslegerForward := FALSE;
        cmdAuslegerBackward := FALSE;
        cmdConveyorForward := FALSE;

        IF HRL_LS_innen THEN
            step := 70;
        END_IF;


    70:
        Busy := TRUE;

        cmdHorizontal := FALSE;
        cmdVertical := FALSE;
        cmdAuslegerForward := FALSE;
        cmdAuslegerBackward := FALSE;
        cmdConveyorForward := TRUE;

        REQ_CB_forwards := fbConveyorForward.DigitalOutputControl_01;

        IF REQ_CB_forwards AND REQ_CB_backwards THEN
            Error := TRUE;
            ErrorId := 206;
            step := 900;
        END_IF;

        IF fbConveyorForward.ResetMethodCall THEN
            cmdConveyorForward := FALSE;
            step := 100;
        END_IF;


    100:
        REQ_CB_forwards := FALSE;
        REQ_CB_backwards := FALSE;

        REQ_RGB_Forwards := FALSE;
        REQ_RGB_Backwards := FALSE;

        REQ_RGB_VerticalDown := FALSE;
        REQ_RGB_VerticalUp := FALSE;

        REQ_RGB_HorizontalForward := FALSE;
        REQ_RGB_HorizontalBackward := FALSE;

        cmdHorizontal := FALSE;
        cmdVertical := FALSE;
        cmdAuslegerForward := FALSE;
        cmdAuslegerBackward := FALSE;
        cmdConveyorForward := FALSE;

        Busy := FALSE;
        Done := TRUE;
        Error := FALSE;
        ErrorId := 0;

        jobRunning := FALSE;
        jobFinished := TRUE;

        MethodCall_Auslagern := FALSE;

        step := 0;


    900:
        REQ_CB_forwards := FALSE;
        REQ_CB_backwards := FALSE;

        REQ_RGB_Forwards := FALSE;
        REQ_RGB_Backwards := FALSE;

        REQ_RGB_VerticalDown := FALSE;
        REQ_RGB_VerticalUp := FALSE;

        REQ_RGB_HorizontalForward := FALSE;
        REQ_RGB_HorizontalBackward := FALSE;

        cmdHorizontal := FALSE;
        cmdVertical := FALSE;
        cmdAuslegerForward := FALSE;
        cmdAuslegerBackward := FALSE;
        cmdConveyorForward := FALSE;

        Busy := FALSE;
        Done := FALSE;

        jobRunning := FALSE;
        jobFinished := TRUE;

        MethodCall_Auslagern := FALSE;

        // Error und ErrorId absichtlich stehen lassen
        step := 0;

ELSE
    REQ_CB_forwards := FALSE;
    REQ_CB_backwards := FALSE;

    REQ_RGB_Forwards := FALSE;
    REQ_RGB_Backwards := FALSE;

    REQ_RGB_VerticalDown := FALSE;
    REQ_RGB_VerticalUp := FALSE;

    REQ_RGB_HorizontalForward := FALSE;
    REQ_RGB_HorizontalBackward := FALSE;

    cmdHorizontal := FALSE;
    cmdVertical := FALSE;
    cmdAuslegerForward := FALSE;
    cmdAuslegerBackward := FALSE;
    cmdConveyorForward := FALSE;

    Busy := FALSE;
    Done := FALSE;
    Error := TRUE;
    ErrorId := 998;

    jobRunning := FALSE;
    jobFinished := TRUE;

    MethodCall_Auslagern := FALSE;

    step := 0;
END_CASE;

CurrentStep := step;

                

{attribute 'TcRpcEnable' := '1'}
METHOD Abort : HRESULT
VAR_INPUT
    hdl : UDINT;
END_VAR
                        callCounterAbort := callCounterAbort + 1;

bAbortRequest := TRUE;

Abort := 0;
                      
END_METHOD

{attribute 'TcRpcEnable' := '1'}
METHOD CheckState : HRESULT
VAR_INPUT
    hdl : UDINT;
END_VAR

VAR_OUTPUT
    bBusy : BOOL;
    State : UDINT;
    IsDone : BOOL;
    HasError : BOOL;
    ErrorCode : UDINT;
END_VAR
                        callCounterCheckState := callCounterCheckState + 1;

bBusy := jobRunning;
State := CurrentStep;
IsDone := jobFinished;
HasError := Error;
ErrorCode := ErrorId;

CheckState := 0;
                      
END_METHOD

{attribute 'TcRpcEnable' := '1'}
METHOD Start : HRESULT
VAR_INPUT
    MethodCall : BOOL;

    HorizontalShelf_I1 : UDINT;
    HorizontalShelf_I2 : UDINT;
    VerticalShelf_I1 : UDINT;
    VerticalShelf_I2 : UDINT;

    HorizontalTransfer_I1 : UDINT;
    HorizontalTransfer_I2 : UDINT;
    VerticalTransfer_I1 : UDINT;
    VerticalTransfer_I2 : UDINT;

    Timeout : TIME;
END_VAR

VAR_OUTPUT
    hdl : UDINT;
END_VAR
                        callCounterStart := callCounterStart + 1;

IF NOT jobRunning THEN
	 IF MethodCall THEN
        OPCUA.lastExecutedProcess := 'HRL_NMethod_Auslagern';
        OPCUA.lastExecutedSkill := 'HRL_NMethod_Auslagern';
    END_IF;
    MethodCall_Auslagern := MethodCall;

    TargetHorizontalShelf_I1 := HorizontalShelf_I1;
    TargetHorizontalShelf_I2 := HorizontalShelf_I2;
    TargetVerticalShelf_I1 := VerticalShelf_I1;
    TargetVerticalShelf_I2 := VerticalShelf_I2;

    TargetHorizontalTransfer_I1 := HorizontalTransfer_I1;
    TargetHorizontalTransfer_I2 := HorizontalTransfer_I2;
    TargetVerticalTransfer_I1 := VerticalTransfer_I1;
    TargetVerticalTransfer_I2 := VerticalTransfer_I2;

    IF Timeout > T#0MS THEN
        WatchdogTime := Timeout;
    ELSE
        WatchdogTime := T#15S;
    END_IF;

    // Neuer Auftrag löscht alten Abschlussstatus
    jobFinished := FALSE;
    Done := FALSE;
    Error := FALSE;
    ErrorId := 0;

    hdl := 1;
    Start := 0;
ELSE
    hdl := 0;
    Start := 16#800700AA;
END_IF;
                      
END_METHOD
END_FUNCTION_BLOCK

{attribute 'OPC.UA.DA.JobMethod' := 'JobMethode_HorizontalMove'}
FUNCTION_BLOCK HRL_RGB_AS_HorizontalMoveEncoders
VAR
	AlwaysTrue : BOOL := TRUE;
	// Used for debugging purposes to display InputArguments of method call
	MethodCall_HorizontalMove : BOOL := FALSE; // used to store InputArg "MethodCall" from Start() method
	ResetMethodCall	: BOOL := FALSE;	
	DirectionHorizontal : BOOL;
	EncoderTargetPosition01 : UDINT;
	EncoderTargetPosition02 : UDINT;
	TSR: BOOL;
	callCounterStart : ULINT; // counts how many times the Start() method has been called
	callCounterCheckState : ULINT; // counts how many times the CheckState() method has been called
	callCounterAbort : ULINT; // counts how many times the Abort() method has been called
	
	// Variables to determine if a job has been started (Start() method has been called) or finished
	jobRunning : BOOL;
	jobFinished : BOOL;

	// State machine variable
	state : UDINT;
	
	// FB Intatziation Variable
	HRL_RGB_HorizontalMoveWithEncoder : AxisControl_Encoder;
END_VAR
	
VAR_INPUT
	ESS						: BOOL;
	TouchSensor01 			: BOOL;
	EncoderStartPosition01 	: UDINT;
	EncoderStartPosition02 	: UDINT;
	TOF_Time_TSR 			: TIME;
	AutomaticMode			: BOOL;
END_VAR

VAR_OUTPUT
	DO_MovingHorizontalRGB_01 : BOOL;
	DO_MovingHorizontalRGB_02 : BOOL;
END_VAR

                  HRL_RGB_HorizontalMoveWithEncoder(
    MethodCall := MethodCall_HorizontalMove,
    EmergencyStopSignal := ESS,
    Direction := DirectionHorizontal,
    InitStateDrive_Input := FALSE,
    DI01 := TouchSensor01,
    DI02_EncoderStart01 := EncoderStartPosition01,
    DI03_EncoderTarget01 := EncoderTargetPosition01,
    DI04_EncoderStart02 := EncoderStartPosition02,
    DI05_EncoderTarget02 := EncoderTargetPosition02,
    TouchSensorRelief := TSR,
    TOF_Time_MotorControl := T#0MS,
    TOF_Time_TouchSensorRelief := TOF_Time_TSR,
    OperatingMode := AutomaticMode
);
DO_MovingHorizontalRGB_01 := HRL_RGB_HorizontalMoveWithEncoder.DigitalOutputControl_01;
                

{attribute 'TcRpcEnable' := '1'}
METHOD Abort : HRESULT
VAR_INPUT
	hdl : UDINT; // Do not change, used by server.
END_VAR
                        callCounterAbort := callCounterAbort + 1;
                      
END_METHOD

{attribute 'TcRpcEnable' := '1'}
METHOD CheckState : HRESULT
VAR_INPUT
	hdl : UDINT; // Do not change, used by server.
END_VAR
VAR_OUTPUT
	bBusy : BOOL; // Do not change. Used by server to find out if the job is finished
	
	// List of OutputArguments for OPC UA method, may be customized
	State : BOOL; // Abgeschlossener MethodCall
	MethodCall: BOOL; //Input Recall
END_VAR
                        callCounterCheckState := callCounterCheckState + 1;
IF NOT jobFinished THEN
	bBusy := TRUE; // job is not finished yet
	CheckState := 0; // no error
ELSE
	bBusy := FALSE; // job is finished
	CheckState := 0; // done, no error occured during execution (OPC UA StatusCode "GOOD")
	jobFinished := FALSE;
	State := ResetMethodCall;
	MethodCall := MethodCall_HorizontalMove;
END_IF
                      
END_METHOD

{attribute 'TcRpcEnable' := '1'}
METHOD Start : HRESULT
VAR_INPUT
	// List of InputArguments for OPC UA method, may be customized
	MethodCall : BOOL; // some description
	MovementDirection : BOOL;
	EncoderPositionHorizontal_01 : UDINT;
	EncoderPositionHorizontal_02 : UDINT;
	TouchSensorRelief : BOOL;
END_VAR
VAR_OUTPUT
	hdl : UDINT; // Do not change, used by server.
END_VAR
                        callCounterStart := callCounterStart + 1;

MethodCall_HorizontalMove := MethodCall;
DirectionHorizontal := MovementDirection;
EncoderTargetPosition01 := EncoderPositionHorizontal_01;
EncoderTargetPosition02 := EncoderPositionHorizontal_02;
TSR := TouchSensorRelief;

jobRunning := TRUE;
Start := 0; // no error occured, e.g. while parsing the input arguments (0 = OPC UA StatusCode "GOOD")
                      
END_METHOD
END_FUNCTION_BLOCK

{attribute 'OPC.UA.DA.JobMethod' := 'JobMethode_HorizontalMove'}
FUNCTION_BLOCK HRL_RGB_AS_HorizontalMoveSensors
VAR
	AlwaysTrue : BOOL := TRUE;
	// Used for debugging purposes to display InputArguments of method call
	MethodCall_HorizontalMove : BOOL := FALSE; // used to store InputArg "MethodCall" from Start() method
	ResetMethodCall	: BOOL := FALSE;	
	DirectionHorizontal : BOOL; // defines movement direction
	TSR : BOOL; // Variable that is needed to perform the relief of the touch sensor
	callCounterStart : ULINT; // counts how many times the Start() method has been called
	callCounterCheckState : ULINT; // counts how many times the CheckState() method has been called
	callCounterAbort : ULINT; // counts how many times the Abort() method has been called
	
	// Variables to determine if a job has been started (Start() method has been called) or finished
	jobRunning : BOOL;
	jobFinished : BOOL;

	// State machine variable
	state : UDINT;
	
	// FB Intatziation Variable
	HRL_RGB_HorizontalMove : AxisControl_MultipleInputSensors;
END_VAR
	
VAR_INPUT
	ESS				: BOOL;
	TouchSensor01 	: BOOL;
	TouchSensor02 	: BOOL;
	TOF_Time_TSR 	: TIME;
	AutomaticMode	: BOOL;
END_VAR

VAR_OUTPUT
	DO_MovingHorizontalRGB_01 : BOOL;
	DO_MovingHorizontalRGB_02 : BOOL;
END_VAR

                  HRL_RGB_HorizontalMove(
    MethodCall := MethodCall_HorizontalMove,
    EmergencyStopSignal := ESS,
    Direction := DirectionHorizontal,
    InitStateDrive_Input := FALSE,
    DI01 := TouchSensor01,
    DI02 := TouchSensor02,
    TouchSensorRelief := TSR,
    TOF_Time_MotorControl := T#0MS,
    TOF_Time_TouchSensorRelief := TOF_Time_TSR,
    OperatingMode := AutomaticMode
);
DO_MovingHorizontalRGB_01 := HRL_RGB_HorizontalMove.DigitalOutputControl_01;


                

{attribute 'TcRpcEnable' := '1'}
METHOD Abort : HRESULT
VAR_INPUT
	hdl : UDINT; // Do not change, used by server.
END_VAR
                        callCounterAbort := callCounterAbort + 1;
                      
END_METHOD

{attribute 'TcRpcEnable' := '1'}
METHOD CheckState : HRESULT
VAR_INPUT
	hdl : UDINT; // Do not change, used by server.
END_VAR
VAR_OUTPUT
	bBusy : BOOL; // Do not change. Used by server to find out if the job is finished
	
	// List of OutputArguments for OPC UA method, may be customized
	State : BOOL; // Abgeschlossener MethodCall
	MethodCall: BOOL; //Input Recall
END_VAR
                        callCounterCheckState := callCounterCheckState + 1;
IF NOT jobFinished THEN
	bBusy := TRUE; // job is not finished yet
	CheckState := 0; // no error
ELSE
	bBusy := FALSE; // job is finished
	CheckState := 0; // done, no error occured during execution (OPC UA StatusCode "GOOD")
	jobFinished := FALSE;
	State := ResetMethodCall;
	MethodCall := MethodCall_HorizontalMove;
END_IF
                      
END_METHOD

{attribute 'TcRpcEnable' := '1'}
METHOD Start : HRESULT
VAR_INPUT
	// List of InputArguments for OPC UA method, may be customized
	MethodCall : BOOL; // some description
	MovementDirection : BOOL;
	TouchSensorRelief : BOOL;
END_VAR
VAR_OUTPUT
	hdl : UDINT; // Do not change, used by server.
END_VAR
                        callCounterStart := callCounterStart + 1;

MethodCall_HorizontalMove := MethodCall;
DirectionHorizontal := MovementDirection;
TSR := TouchSensorRelief;

jobRunning := TRUE;
Start := 0; // OPC UA StatusCode GOOD
                      
END_METHOD
END_FUNCTION_BLOCK

{attribute 'OPC.UA.DA.JobMethod' := 'JobMethode_VerticalMove'}
FUNCTION_BLOCK HRL_RGB_AS_VerticalMoveEncoders
VAR
	AlwaysTrue : BOOL := TRUE;
	// Used for debugging purposes to display InputArguments of method call
	MethodCall_VerticalMove : BOOL := FALSE; // used to store InputArg "MethodCall" from Start() method
	ResetMethodCall	: BOOL := FALSE;
	DirectionVertical : BOOL;
	EncoderTargetPosition01 : UDINT;
	EncoderTargetPosition02 : UDINT;
	TSR : BOOL;
	callCounterStart : ULINT; // counts how many times the Start() method has been called
	callCounterCheckState : ULINT; // counts how many times the CheckState() method has been called
	callCounterAbort : ULINT; // counts how many times the Abort() method has been called
	
	// Variables to determine if a job has been started (Start() method has been called) or finished
	jobRunning : BOOL;
	jobFinished : BOOL;

	// State machine variable
	state : UDINT;
	
	// FB Intatziation Variable
	HRL_RGB_VerticalMoveWithEncoder : AxisControl_Encoder;
END_VAR
	
VAR_INPUT
	ESS: BOOL;
	TouchSensor01 : BOOL;
	EncoderStartPosition01 : UDINT;
	EncoderStartPosition02 : UDINT;
	TOF_TSR_TIME : TIME;
	AutomaticMode: BOOL;
END_VAR

VAR_OUTPUT
	DO_MovingVerticalRGB_01 : BOOL;
	DO_MovingVerticalRGB_02 : BOOL;
END_VAR

                  HRL_RGB_VerticalMoveWithEncoder(
    MethodCall := MethodCall_VerticalMove,
    EmergencyStopSignal := ESS,
    Direction := DirectionVertical,
    InitStateDrive_Input := FALSE,
    DI01 := TouchSensor01,
    DI02_EncoderStart01 := EncoderStartPosition01,
    DI03_EncoderTarget01 := EncoderTargetPosition01,
    DI04_EncoderStart02 := EncoderStartPosition02,
    DI05_EncoderTarget02 := EncoderTargetPosition02,
    TouchSensorRelief := TSR,
    TOF_Time_MotorControl := T#0MS,
    TOF_Time_TouchSensorRelief := TOF_TSR_TIME,
    OperatingMode := AutomaticMode
);
DO_MovingVerticalRGB_01 := HRL_RGB_VerticalMoveWithEncoder.DigitalOutputControl_01;

                

{attribute 'TcRpcEnable' := '1'}
METHOD Abort : HRESULT
VAR_INPUT
	hdl : UDINT; // Do not change, used by server.
END_VAR
                        callCounterAbort := callCounterAbort + 1;
                      
END_METHOD

{attribute 'TcRpcEnable' := '1'}
METHOD CheckState : HRESULT
VAR_INPUT
	hdl : UDINT; // Do not change, used by server.
END_VAR
VAR_OUTPUT
	bBusy : BOOL; // Do not change. Used by server to find out if the job is finished
	
	// List of OutputArguments for OPC UA method, may be customized
	State : BOOL; // Abgeschlossener MethodCall
	MethodCall: BOOL; //Input Recall
END_VAR
                        callCounterCheckState := callCounterCheckState + 1;
IF NOT jobFinished THEN
	bBusy := TRUE; // job is not finished yet
	CheckState := 0; // no error
ELSE
	bBusy := FALSE; // job is finished
	CheckState := 0; // done, no error occured during execution (OPC UA StatusCode "GOOD")
	jobFinished := FALSE;
	State := ResetMethodCall;
	MethodCall := MethodCall_VerticalMove;
END_IF
                      
END_METHOD

{attribute 'TcRpcEnable' := '1'}
METHOD Start : HRESULT
VAR_INPUT
	// List of InputArguments for OPC UA method, may be customized
	MethodCall : BOOL; // some description
	MovementDirection : BOOL;
	EncoderPositionVertical_01 : UDINT;
	EncoderPositionVertical_02 : UDINT;
	TouchSensorRelief : BOOL;
END_VAR
VAR_OUTPUT
	hdl : UDINT; // Do not change, used by server.
END_VAR
                        callCounterStart := callCounterStart + 1;

MethodCall_VerticalMove := MethodCall;
DirectionVertical := MovementDirection;
EncoderTargetPosition01 := EncoderPositionVertical_01;
EncoderTargetPosition02 := EncoderPositionVertical_02;
TSR := TouchSensorRelief;

jobRunning := TRUE;
Start := 0; // no error occured, e.g. while parsing the input arguments (0 = OPC UA StatusCode "GOOD")
                      
END_METHOD
END_FUNCTION_BLOCK

{attribute 'OPC.UA.DA.JobMethod' := 'JobMethode_HorizontalMove'}
FUNCTION_BLOCK MBS_CB_AS_HorizontalMove
VAR
	AlwaysTrue : BOOL := TRUE;
	// Used for debugging purposes to display InputArguments of method call
	MethodCall_HorizontalMove : BOOL := FALSE; // used to store InputArg "MethodCall" from Start() method
	ResetMethodCall	: BOOL := FALSE;	
	DirectionHorizontal : STRING; // defines movement direction
	callCounterStart : ULINT; // counts how many times the Start() method has been called
	callCounterCheckState : ULINT; // counts how many times the CheckState() method has been called
	callCounterAbort : ULINT; // counts how many times the Abort() method has been called
	
	// Variables to determine if a job has been started (Start() method has been called) or finished
	jobRunning : BOOL;
	jobFinished : BOOL;

	// State machine variable
	state : UDINT;
	
	// FB Intatziation Variable
	MBS_CB_HorizontalMove : AxisControl_MultipleInputSensors;
END_VAR
	
VAR_INPUT
	ESS: BOOL;
	TouchSensor_01 : BOOL;
	LightSensor_01 : BOOL;
	TOF_Time_MotorControl : TIME;
	AutomaticMode: BOOL;
END_VAR

VAR_OUTPUT
	DO_MovingHorizontalCB_01 : BOOL;
END_VAR

                  MBS_CB_HorizontalMove(
    MethodCall := MethodCall_HorizontalMove,
    EmergencyStopSignal := ESS,
    Direction := DirectionHorizontal,
    InitStateDrive_Input := ,
    DI01 := TouchSensor_01,
    DI02 := LightSensor_01,
    TouchSensorRelief := ,
    TOF_Time_MotorControl := TOF_Time_MotorControl,
    TOF_Time_TouchSensorRelief := ,
    OperatingMode := AutomaticMode
);
DO_MovingHorizontalCB_01 := MBS_CB_HorizontalMove.DigitalOutputControl_01;
                

{attribute 'TcRpcEnable' := '1'}
METHOD Abort : HRESULT
VAR_INPUT
	hdl : UDINT; // Do not change, used by server.
END_VAR
                        callCounterAbort := callCounterAbort + 1;
                      
END_METHOD

{attribute 'TcRpcEnable' := '1'}
METHOD CheckState : HRESULT
VAR_INPUT
	hdl : UDINT; // Do not change, used by server.
END_VAR
VAR_OUTPUT
	bBusy : BOOL; // Do not change. Used by server to find out if the job is finished
	
	// List of OutputArguments for OPC UA method, may be customized
	State : BOOL; // Abgeschlossener MethodCall
	MethodCall: BOOL; //Input Recall
END_VAR
                        callCounterCheckState := callCounterCheckState + 1;
IF NOT jobFinished THEN
	bBusy := TRUE; // job is not finished yet
	CheckState := 0; // no error
ELSE
	bBusy := FALSE; // job is finished
	CheckState := 0; // done, no error occured during execution (OPC UA StatusCode "GOOD")
	jobFinished := FALSE;
	State := ResetMethodCall;
	MethodCall := MethodCall_HorizontalMove;
END_IF
                      
END_METHOD

{attribute 'TcRpcEnable' := '1'}
METHOD Start : HRESULT
VAR_INPUT
	// List of InputArguments for OPC UA method, may be customized
	MethodCall : BOOL; // some description
	DirectionPoint : STRING;	
END_VAR
VAR_OUTPUT
	hdl : UDINT; // Do not change, used by server.
END_VAR
                        callCounterStart := callCounterStart + 1;

MethodCall_HorizontalMove := MethodCall;
DirectionHorizontal := DirectionPoint;

jobRunning := TRUE;
Start := 0; // no error occured, e.g. while parsing the input arguments (0 = OPC UA StatusCode "GOOD")
                      
END_METHOD
END_FUNCTION_BLOCK

{attribute 'OPC.UA.DA.JobMethod' := 'JobMethode_CompressorControl'}
FUNCTION_BLOCK MBS_DmPD_AS_HorizontalMove
VAR
	AlwaysTrue : BOOL := TRUE;
	// Used for debugging purposes to display InputArguments of method call
	MethodCall_CompressorControl : BOOL := FALSE; // used to store InputArg "MethodCall" from Start() method
	ResetMethodCall	: BOOL := FALSE;
	DestinationVertical : STRING;
	PowerOFF_SelfSet : BOOL;
	PowerOFFDelay_SelfSet : TIME;
	callCounterStart : ULINT; // counts how many times the Start() method has been called
	callCounterCheckState : ULINT; // counts how many times the CheckState() method has been called
	callCounterAbort : ULINT; // counts how many times the Abort() method has been called
	
	// Variables to determine if a job has been started (Start() method has been called) or finished
	jobRunning : BOOL;
	jobFinished : BOOL;

	// State machine variable
	state : UDINT;
	
	//Variablen des Transport FBs
	MBS_DmPD_VerticalMove : CompressorControl;
END_VAR
	
VAR_INPUT
	ESS: BOOL;
	TouchSensor_01 : BOOL;
	TON_PowerOnDelay_Compressor : TIME;
	TON_PowerOnDelay_Valve : TIME;
	AutomaticMode: BOOL;
END_VAR

VAR_OUTPUT
	DO_ControlCompressorDmPD_01 : BOOL;
	DO_ControlValveDmPD_02 : BOOL;
END_VAR

                  MBS_DmPD_VerticalMove(
    MethodCall := MethodCall_CompressorControl,
    EmergencyStopSignal := ESS,
    Destination := DestinationVertical,
    InitStateDrive_Input := ,
    DI01 := TouchSensor_01,
    DI02 := ,
    DI03_EncoderStart01 := ,
    DI04_EncoderStart02 := ,
    DI05_EncoderStart03 := ,
    DI06_EncoderStart04 := ,
    DI07_EncoderStart05 := ,
    DI08_EncoderStart06 := ,
    DI09_EncoderTarget01 := ,
    DI10_EncoderTarget02 := ,
    DI11_EncoderTarget03 := ,
    DI12_EncoderTarget04 := ,
    DI13_EncoderTarget05 := ,
    DI14_EncoderTarget06 := ,
    PowerOFF_SelfSet := PowerOFF_SelfSet,
    TON_Time_PowerOFFSelfSet := PowerOFFDelay_SelfSet,
    TON_Time_Compressor := TON_PowerOnDelay_Compressor,
    TON_Time_Valve := TON_PowerOnDelay_Valve,
    OperatingMode := AutomaticMode
);
DO_ControlCompressorDmPD_01 := MBS_DmPD_VerticalMove.DigitalOutputControl_01;

                

{attribute 'TcRpcEnable' := '1'}
METHOD Abort : HRESULT
VAR_INPUT
	hdl : UDINT; // Do not change, used by server.
END_VAR
                        callCounterAbort := callCounterAbort + 1;
                      
END_METHOD

{attribute 'TcRpcEnable' := '1'}
METHOD CheckState : HRESULT
VAR_INPUT
	hdl : UDINT; // Do not change, used by server.
END_VAR
VAR_OUTPUT
	bBusy : BOOL; // Do not change. Used by server to find out if the job is finished
	
	// List of OutputArguments for OPC UA method, may be customized
	State : BOOL; // Abgeschlossener MethodCall
	MethodCall: BOOL; //Input Recall
END_VAR
                        callCounterCheckState := callCounterCheckState + 1;
IF NOT jobFinished THEN
	bBusy := TRUE; // job is not finished yet
	CheckState := 0; // no error
ELSE
	bBusy := FALSE; // job is finished
	CheckState := 0; // done, no error occured during execution (OPC UA StatusCode "GOOD")
	jobFinished := FALSE;
	State := ResetMethodCall;
	MethodCall := MethodCall_CompressorControl;
END_IF
                      
END_METHOD

{attribute 'TcRpcEnable' := '1'}
METHOD Start : HRESULT
VAR_INPUT
	// List of InputArguments for OPC UA method, may be customized
	MethodCall : BOOL; // some description
	DestinationPoint : STRING;
	SelfSetPowerOff : BOOL;
	SelfSetPowerOffDelay : TIME;	
END_VAR
VAR_OUTPUT
	hdl : UDINT; // Do not change, used by server.
END_VAR
                        callCounterStart := callCounterStart + 1;

MethodCall_CompressorControl := MethodCall;
DestinationVertical := DestinationPoint;
PowerOFF_SelfSet := SelfSetPowerOff;
PowerOFFDelay_SelfSet := SelfSetPowerOffDelay;

jobRunning := TRUE;
Start := 0; // no error occured, e.g. while parsing the input arguments (0 = OPC UA StatusCode "GOOD")
                      
END_METHOD
END_FUNCTION_BLOCK

{attribute 'OPC.UA.DA.JobMethod' := 'JobMethode_RotationMove'}
FUNCTION_BLOCK MBS_DmPD_AS_RotationMove
VAR
	AlwaysTrue : BOOL := TRUE;
	// Used for debugging purposes to display InputArguments of method call
	MethodCall_RotationMove : BOOL := FALSE; // used to store InputArg "MethodCall" from Start() method
	ResetMethodCall : BOOL := FALSE;
	DirectionRotation : STRING;
	callCounterStart : ULINT; // counts how many times the Start() method has been called
	callCounterCheckState : ULINT; // counts how many times the CheckState() method has been called
	callCounterAbort : ULINT; // counts how many times the Abort() method has been called
	
	// Variables to determine if a job has been started (Start() method has been called) or finished
	jobRunning : BOOL;
	jobFinished : BOOL;

	// State machine variable
	state : UDINT;
	
	//Variablen des Transport FBs
	MBS_DmPD_RotationMove : AxisControl_MultipleInputSensors;
END_VAR
	
VAR_INPUT
	ESS: BOOL;
	TouchSensor_01 : BOOL;
	TouchSensor_02 : BOOL;
	AutomaticMode: BOOL;
END_VAR

VAR_OUTPUT
	DO_MovingRotationPmPD_01 : BOOL;
	DO_MovingRotationPmPD_02 : BOOL;
END_VAR

                  MBS_DmPD_RotationMove(
    MethodCall := MethodCall_RotationMove,
    EmergencyStopSignal := ESS,
    Direction := DirectionRotation,
    InitStateDrive_Input := ,
    DI01 := TouchSensor_01,
    DI02 := TouchSensor_02,
    TouchSensorRelief := ,
    TOF_Time_MotorControl := ,
    TOF_Time_TouchSensorRelief := ,
    OperatingMode := AutomaticMode
);
DO_MovingRotationPmPD_01 := MBS_DmPD_RotationMove.DigitalOutputControl_01;

                

{attribute 'TcRpcEnable' := '1'}
METHOD Abort : HRESULT
VAR_INPUT
	hdl : UDINT; // Do not change, used by server.
END_VAR
                        callCounterAbort := callCounterAbort + 1;
                      
END_METHOD

{attribute 'TcRpcEnable' := '1'}
METHOD CheckState : HRESULT
VAR_INPUT
	hdl : UDINT; // Do not change, used by server.
END_VAR
VAR_OUTPUT
	bBusy : BOOL; // Do not change. Used by server to find out if the job is finished
	
	// List of OutputArguments for OPC UA method, may be customized
	State : BOOL; // Abgeschlossener MethodCall
	MethodCall: BOOL; //Input Recall
END_VAR
                        callCounterCheckState := callCounterCheckState + 1;
IF NOT jobFinished THEN
	bBusy := TRUE; // job is not finished yet
	CheckState := 0; // no error
ELSE
	bBusy := FALSE; // job is finished
	CheckState := 0; // done, no error occured during execution (OPC UA StatusCode "GOOD")
	jobFinished := FALSE;
	State := ResetMethodCall;
	MethodCall := MethodCall_RotationMove;
END_IF
                      
END_METHOD

{attribute 'TcRpcEnable' := '1'}
METHOD Start : HRESULT
VAR_INPUT
	// List of InputArguments for OPC UA method, may be customized
	MethodCall : BOOL; // some description
	DirectionPoint : STRING;		
END_VAR
VAR_OUTPUT
	hdl : UDINT; // Do not change, used by server.
END_VAR
                        callCounterStart := callCounterStart + 1;

MethodCall_RotationMove := MethodCall;
DirectionRotation := DirectionPoint;

jobRunning := TRUE;
Start := 0; // no error occured, e.g. while parsing the input arguments (0 = OPC UA StatusCode "GOOD")
                      
END_METHOD
END_FUNCTION_BLOCK

{attribute 'OPC.UA.DA.JobMethod' := 'JobMethode_HardeningProcess'}
FUNCTION_BLOCK MBS_MR01_AS_HardeningProcess
VAR
	AlwaysTrue : BOOL := TRUE;
	// Used for debugging purposes to display InputArguments of method call
	MethodCall_HardeningProcess : BOOL := FALSE; // used to store InputArg "MethodCall" from Start() method
	ResetMethodCall	: BOOL := FALSE;
	ProcessingTime_HardeningProcess : TIME;
	callCounterStart : ULINT; // counts how many times the Start() method has been called
	callCounterCheckState : ULINT; // counts how many times the CheckState() method has been called
	callCounterAbort : ULINT; // counts how many times the Abort() method has been called
	
	// Variables to determine if a job has been started (Start() method has been called) or finished
	jobRunning : BOOL;
	jobFinished : BOOL;

	// State machine variable
	state : UDINT;
	
	//Variablen des FBs
	MBS_MR01_HardeningProcess : HardeningProcess;
END_VAR
	
VAR_INPUT
	ESS: BOOL;
	LightSensor_01 : BOOL;
	AutomaticMode : BOOL;
END_VAR

VAR_OUTPUT
	DO_HardeningProcessControlMR01 : BOOL;
END_VAR

                  MBS_MR01_HardeningProcess(
    MethodCall := MethodCall_HardeningProcess,
    EmergencyStopSignal := ESS,
    InitStateDrive_Input := ,
    DI01 := LightSensor_01,
    TOF_Time_HardeningTime := ProcessingTime_HardeningProcess,
    OperatingMode := AutomaticMode
);
DO_HardeningProcessControlMR01 := MBS_MR01_HardeningProcess.DigitalOutputControl_01;
                

{attribute 'TcRpcEnable' := '1'}
METHOD Abort : HRESULT
VAR_INPUT
	hdl : UDINT; // Do not change, used by server.
END_VAR
                        callCounterAbort := callCounterAbort + 1;
                      
END_METHOD

{attribute 'TcRpcEnable' := '1'}
METHOD CheckState : HRESULT
VAR_INPUT
	hdl : UDINT; // Do not change, used by server.
END_VAR
VAR_OUTPUT
	bBusy : BOOL; // Do not change. Used by server to find out if the job is finished
	
	// List of OutputArguments for OPC UA method, may be customized
	State : BOOL; // Abgeschlossener MethodCall
	MethodCall: BOOL; //Input Recall
END_VAR
                        callCounterCheckState := callCounterCheckState + 1;
IF NOT jobFinished THEN
	bBusy := TRUE; // job is not finished yet
	CheckState := 0; // no error
ELSE
	bBusy := FALSE; // job is finished
	CheckState := 0; // done, no error occured during execution (OPC UA StatusCode "GOOD")
	jobFinished := FALSE;
	State := ResetMethodCall;
	MethodCall := MethodCall_HardeningProcess;
END_IF
                      
END_METHOD

{attribute 'TcRpcEnable' := '1'}
METHOD Start : HRESULT
VAR_INPUT
	// List of InputArguments for OPC UA method, may be customized
	MethodCall : BOOL; // some description
	ProcessingTime : TIME;
END_VAR
VAR_OUTPUT
	hdl : UDINT; // Do not change, used by server.
END_VAR
                        callCounterStart := callCounterStart + 1;

MethodCall_HardeningProcess := MethodCall;
ProcessingTime_HardeningProcess := ProcessingTime;

jobRunning := TRUE;
Start := 0; // no error occured, e.g. while parsing the input arguments (0 = OPC UA StatusCode "GOOD")
                      
END_METHOD
END_FUNCTION_BLOCK

{attribute 'OPC.UA.DA.JobMethod' := 'JobMethode_HorizontalMove'}
FUNCTION_BLOCK MBS_MR01_AS_HorizontalMoveSensors
VAR
	AlwaysTrue : BOOL := TRUE;
	// Used for debugging purposes to display InputArguments of method call
	MethodCall_HorizontalMove : BOOL := FALSE; // used to store InputArg "MethodCall" from Start() method
	ResetMethodCall : BOOL := FALSE;
	DirectionHorizontal : STRING; // defines movement direction
	TSR : BOOL; // Variable that is needed to perform the relief of the touch sensor
	callCounterStart : ULINT; // counts how many times the Start() method has been called
	callCounterCheckState : ULINT; // counts how many times the CheckState() method has been called
	callCounterAbort : ULINT; // counts how many times the Abort() method has been called
	
	// Variables to determine if a job has been started (Start() method has been called) or finished
	jobRunning : BOOL;
	jobFinished : BOOL;

	// State machine variable
	state : UDINT;
	
	//Variablen des Transport FBs
	MBS_MR01_HorizontalMove : AxisControl_MultipleInputSensors;
END_VAR
	
VAR_INPUT
	ESS: BOOL;
	TouchSensor_01 : BOOL;
	TouchSensor_02 : BOOL;
	TOF_Time_TSR : TIME;
	AutomaticMode : BOOL;
END_VAR

VAR_OUTPUT
	DO_MovingHorizontalMR01_01 : BOOL;
	DO_MovingHorizontalMR01_02 : BOOL;
END_VAR

                  (* ST implementation auto-generated from FBD in export.xml *)
MBS_MR01_HorizontalMove(
    MethodCall := MethodCall_HorizontalMove,
    EmergencyStopSignal := ESS,
    Direction := DirectionHorizontal,
    InitStateDrive_Input := ,
    DI01 := TouchSensor_01,
    DI02 := TouchSensor_02,
    TouchSensorRelief := TSR,
    TOF_Time_MotorControl := ,
    TOF_Time_TouchSensorRelief := TOF_Time_TSR,
    OperatingMode := AutomaticMode
);
DO_MovingHorizontalMR01_01 := MBS_MR01_HorizontalMove.DigitalOutputControl_01;

                

{attribute 'TcRpcEnable' := '1'}
METHOD Abort : HRESULT
VAR_INPUT
	hdl : UDINT; // Do not change, used by server.
END_VAR
                        callCounterAbort := callCounterAbort + 1;
                      
END_METHOD

{attribute 'TcRpcEnable' := '1'}
METHOD CheckState : HRESULT
VAR_INPUT
	hdl : UDINT; // Do not change, used by server.
END_VAR
VAR_OUTPUT
	bBusy : BOOL; // Do not change. Used by server to find out if the job is finished
	
	// List of OutputArguments for OPC UA method, may be customized
	State : BOOL; // Abgeschlossener MethodCall
	MethodCall: BOOL; //Input Recall
END_VAR
                        callCounterCheckState := callCounterCheckState + 1;
IF NOT jobFinished THEN
	bBusy := TRUE; // job is not finished yet
	CheckState := 0; // no error
ELSE
	bBusy := FALSE; // job is finished
	CheckState := 0; // done, no error occured during execution (OPC UA StatusCode "GOOD")
	jobFinished := FALSE;
	State := ResetMethodCall;
	MethodCall := MethodCall_HorizontalMove;
END_IF
                      
END_METHOD

{attribute 'TcRpcEnable' := '1'}
METHOD Start : HRESULT
VAR_INPUT
	// List of InputArguments for OPC UA method, may be customized
	MethodCall : BOOL; // some description
	ProcessingTime : TIME;
END_VAR
VAR_OUTPUT
	hdl : UDINT; // Do not change, used by server.
END_VAR
                        callCounterStart := callCounterStart + 1;

MethodCall_HardeningProcess := MethodCall;
ProcessingTime_HardeningProcess := ProcessingTime;

jobRunning := TRUE;
Start := 0; // no error occured, e.g. while parsing the input arguments (0 = OPC UA StatusCode "GOOD")
                      
END_METHOD
END_FUNCTION_BLOCK

{attribute 'OPC.UA.DA.JobMethod' := 'JobMethode_SecuringProcess'}
FUNCTION_BLOCK MBS_MR01_AS_SecuringProcess
VAR
	AlwaysTrue : BOOL := TRUE;
	// Used for debugging purposes to display InputArguments of method call
	MethodCall_SecuringProcess : BOOL := FALSE; // used to store InputArg "MethodCall" from Start() method
	ResetMethodCall	: BOOL := FALSE;	
	SecuringTime : TIME;	//Time for Securing the Workpiece
	SecuringProcessingTime : TIME; //Two Times for Securing the Workpiece (for Secure and Release) + HardeningProcessingTime
	callCounterStart : ULINT; // counts how many times the Start() method has been called
	callCounterCheckState : ULINT; // counts how many times the CheckState() method has been called
	callCounterAbort : ULINT; // counts how many times the Abort() method has been called
	
	// Variables to determine if a job has been started (Start() method has been called) or finished
	jobRunning : BOOL;
	jobFinished : BOOL;

	// State machine variable
	state : UDINT;
	
	//Variablen des FBs
	MBS_MR01_SecuringProcess : SecuringWorkpiece;
END_VAR
	
VAR_INPUT
	ESS: BOOL;
	TouchSensor_01 : BOOL;
	AutomaticMode: BOOL;
END_VAR

VAR_OUTPUT
	DO_SecuringProcessCompressorMR01_01 : BOOL;
	DO_SecuringProcessValveMR01_02 : BOOL;
END_VAR

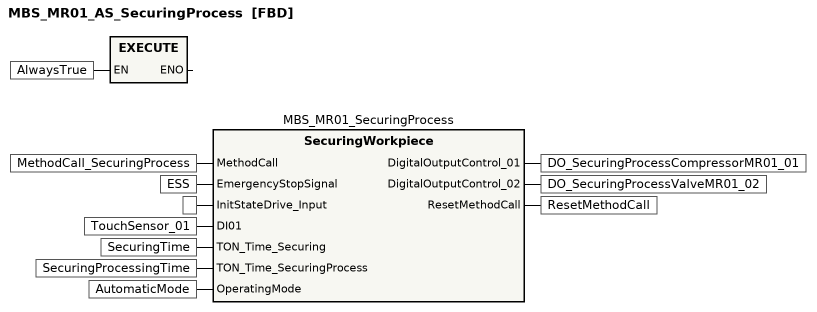
(* FBD diagram, written out as Structured Text *)
IF AlwaysTrue THEN
  CASE state OF
  	0:
  		IF jobRunning THEN
  			state := state + 1;
  		END_IF
  		
  	1:
  		IF ResetMethodCall THEN
  			jobRunning := FALSE;
  			jobFinished := TRUE;
  			state := 0;
  			MethodCall_SecuringProcess := FALSE;
  		END_IF
  		
  END_CASE
END_IF;
MBS_MR01_SecuringProcess(MethodCall := MethodCall_SecuringProcess, EmergencyStopSignal := ESS, InitStateDrive_Input := , DI01 := TouchSensor_01, TON_Time_Securing := SecuringTime, TON_Time_SecuringProcess := SecuringProcessingTime, OperatingMode := AutomaticMode, DigitalOutputControl_02 => DO_SecuringProcessValveMR01_02, ResetMethodCall => ResetMethodCall);
DO_SecuringProcessCompressorMR01_01 := MBS_MR01_SecuringProcess.DigitalOutputControl_01;

{attribute 'TcRpcEnable' := '1'}
METHOD Abort : HRESULT
VAR_INPUT
	hdl : UDINT; // Do not change, used by server.
END_VAR
                        callCounterAbort := callCounterAbort + 1;
                      
END_METHOD

{attribute 'TcRpcEnable' := '1'}
METHOD CheckState : HRESULT
VAR_INPUT
	hdl : UDINT; // Do not change, used by server.
END_VAR
VAR_OUTPUT
	bBusy : BOOL; // Do not change. Used by server to find out if the job is finished
	
	// List of OutputArguments for OPC UA method, may be customized
	State : BOOL; // Abgeschlossener MethodCall
	MethodCall: BOOL; //Input Recall
END_VAR
                        callCounterCheckState := callCounterCheckState + 1;
IF NOT jobFinished THEN
	bBusy := TRUE; // job is not finished yet
	CheckState := 0; // no error
ELSE
	bBusy := FALSE; // job is finished
	CheckState := 0; // done, no error occured during execution (OPC UA StatusCode "GOOD")
	jobFinished := FALSE;
	State := ResetMethodCall;
	MethodCall := MethodCall_SecuringProcess;
END_IF
                      
END_METHOD

{attribute 'TcRpcEnable' := '1'}
METHOD Start : HRESULT
VAR_INPUT
	// List of InputArguments for OPC UA method, may be customized
	MethodCall : BOOL; // some description
	Securing_Time : TIME;
	SecuringProcessing_Time : TIME;
END_VAR
VAR_OUTPUT
	hdl : UDINT; // Do not change, used by server.
END_VAR
                        callCounterStart := callCounterStart + 1;

MethodCall_SecuringProcess := MethodCall;
SecuringTime := Securing_Time;
SecuringProcessingTime := SecuringProcessing_Time;

jobRunning := TRUE;
Start := 0; // no error occured, e.g. while parsing the input arguments (0 = OPC UA StatusCode "GOOD")
                      
END_METHOD
END_FUNCTION_BLOCK

{attribute 'OPC.UA.DA.JobMethod' := 'JobMethode_CuttingProcess'}
FUNCTION_BLOCK MBS_MR02_AS_CuttingProcess
VAR
	AlwaysTrue : BOOL := TRUE;
	// Used for debugging purposes to display InputArguments of method call
	MethodCall_CuttingProcess : BOOL := FALSE; // used to store InputArg "MethodCall" from Start() method
	ResetMethodCall	: BOOL := FALSE;
	ProcessingTime_CuttingProcess : TIME;
	callCounterStart : ULINT; // counts how many times the Start() method has been called
	callCounterCheckState : ULINT; // counts how many times the CheckState() method has been called
	callCounterAbort : ULINT; // counts how many times the Abort() method has been called
	
	// Variables to determine if a job has been started (Start() method has been called) or finished
	jobRunning : BOOL;
	jobFinished : BOOL;

	// State machine variable
	state : UDINT;
	
	//Variablen des FBs
	MBS_MR02_CuttingProcess : CuttingProcess;
END_VAR
	
VAR_INPUT
	ESS: BOOL;
	TouchSensor_01 : BOOL;
	AutomaticMode : BOOL;
END_VAR

VAR_OUTPUT
	DO_CuttingProcessControlMR02 : BOOL;
END_VAR

                  MBS_MR02_CuttingProcess(
    MethodCall := MethodCall_CuttingProcess,
    EmergencyStopSignal := ESS,
    InitStateDrive_Input := ,
    DI01 := TouchSensor_01,
    TOF_Time_CuttingTime := ProcessingTime_CuttingProcess,
    OperatingMode := AutomaticMode
);
DO_CuttingProcessControlMR02 := MBS_MR02_CuttingProcess.DigitalOutputControl_01;

                

{attribute 'TcRpcEnable' := '1'}
METHOD Abort : HRESULT
VAR_INPUT
	hdl : UDINT; // Do not change, used by server.
END_VAR
                        callCounterAbort := callCounterAbort + 1;
                      
END_METHOD

{attribute 'TcRpcEnable' := '1'}
METHOD CheckState : HRESULT
VAR_INPUT
	hdl : UDINT; // Do not change, used by server.
END_VAR
VAR_OUTPUT
	bBusy : BOOL; // Do not change. Used by server to find out if the job is finished
	
	// List of OutputArguments for OPC UA method, may be customized
	State : BOOL; // Abgeschlossener MethodCall
	MethodCall: BOOL; //Input Recall
END_VAR
                        callCounterCheckState := callCounterCheckState + 1;
IF NOT jobFinished THEN
	bBusy := TRUE; // job is not finished yet
	CheckState := 0; // no error
ELSE
	bBusy := FALSE; // job is finished
	CheckState := 0; // done, no error occured during execution (OPC UA StatusCode "GOOD")
	jobFinished := FALSE;
	State := ResetMethodCall;
	MethodCall := MethodCall_CuttingProcess;
END_IF
                      
END_METHOD

{attribute 'TcRpcEnable' := '1'}
METHOD Start : HRESULT
VAR_INPUT
	// List of InputArguments for OPC UA method, may be customized
	MethodCall : BOOL; // some description
	ProcessingTime : TIME;
END_VAR
VAR_OUTPUT
	hdl : UDINT; // Do not change, used by server.
END_VAR
                        callCounterStart := callCounterStart + 1;

MethodCall_CuttingProcess := MethodCall;
ProcessingTime_CuttingProcess := ProcessingTime;

jobRunning := TRUE;
Start := 0; // no error occured, e.g. while parsing the input arguments (0 = OPC UA StatusCode "GOOD")
                      
END_METHOD
END_FUNCTION_BLOCK

{attribute 'OPC.UA.DA.JobMethod' := 'JobMethode_HorizontalMove'}
FUNCTION_BLOCK MBS_VSG_AS_HorizontalMove
VAR
	AlwaysTrue : BOOL := TRUE;
	// Used for debugging purposes to display InputArguments of method call
	MethodCall_HorizontalMove : BOOL := FALSE; // used to store InputArg "MethodCall" from Start() method
	ResetMethodCall	: BOOL := FALSE;
	DirectionHorizontal : STRING; // defines movement direction
	TSR : BOOL;// Variable that is needed to perform the relief of the touch sensor
	callCounterStart : ULINT; // counts how many times the Start() method has been called
	callCounterCheckState : ULINT; // counts how many times the CheckState() method has been called
	callCounterAbort : ULINT; // counts how many times the Abort() method has been called
	
	// Variables to determine if a job has been started (Start() method has been called) or finished
	jobRunning : BOOL;
	jobFinished : BOOL;

	// State machine variable
	state : UDINT;
	
	//Variablen des Transport FBs
	MBS_VSG_HorizontalMove : AxisControl_MultipleInputSensors;
END_VAR
	
VAR_INPUT
	ESS: BOOL;
	TouchSensor_01 : BOOL;
	TouchSensor_02 : BOOL;
	TOF_Time_TSR : TIME;
	AutomaticeMode : BOOL;
END_VAR

VAR_OUTPUT
	DO_HorizontalMoveVSG_01 : BOOL;
	DO_HorizontalMoveVSG_02 : BOOL;
END_VAR

                  MBS_VSG_HorizontalMove(
    MethodCall := MethodCall_HorizontalMove,
    EmergencyStopSignal := ESS,
    Direction := DirectionHorizontal,
    InitStateDrive_Input := ,
    DI01 := TouchSensor_01,
    DI02 := TouchSensor_02,
    TouchSensorRelief := TSR,
    TOF_Time_MotorControl := ,
    TOF_Time_TouchSensorRelief := TOF_Time_TSR,
    OperatingMode := AutomaticeMode
);
DO_HorizontalMoveVSG_01 := MBS_VSG_HorizontalMove.DigitalOutputControl_01;

                

{attribute 'TcRpcEnable' := '1'}
METHOD Abort : HRESULT
VAR_INPUT
	hdl : UDINT; // Do not change, used by server.
END_VAR
                        callCounterAbort := callCounterAbort + 1;
                      
END_METHOD

{attribute 'TcRpcEnable' := '1'}
METHOD CheckState : HRESULT
VAR_INPUT
	hdl : UDINT; // Do not change, used by server.
END_VAR
VAR_OUTPUT
	bBusy : BOOL; // Do not change. Used by server to find out if the job is finished
	
	// List of OutputArguments for OPC UA method, may be customized
	State : BOOL; // Abgeschlossener MethodCall
	MethodCall: BOOL; //Input Recall
END_VAR
                        callCounterCheckState := callCounterCheckState + 1;
IF NOT jobFinished THEN
	bBusy := TRUE; // job is not finished yet
	CheckState := 0; // no error
ELSE
	bBusy := FALSE; // job is finished
	CheckState := 0; // done, no error occured during execution (OPC UA StatusCode "GOOD")
	jobFinished := FALSE;
	State := ResetMethodCall;
	MethodCall := MethodCall_HorizontalMove;
END_IF
                      
END_METHOD

{attribute 'TcRpcEnable' := '1'}
METHOD Start : HRESULT
VAR_INPUT
	// List of InputArguments for OPC UA method, may be customized
	MethodCall : BOOL; // some description
	DirectionPoint : STRING;
	TouchSensorRelief : BOOL;	
END_VAR
VAR_OUTPUT
	hdl : UDINT; // Do not change, used by server.
END_VAR
                        callCounterStart := callCounterStart + 1;

MethodCall_HorizontalMove := MethodCall;
DirectionHorizontal := DirectionPoint;
TSR := TouchSensorRelief;

jobRunning := TRUE;
Start := 0; // no error occured, e.g. while parsing the input arguments (0 = OPC UA StatusCode "GOOD")
                      
END_METHOD
END_FUNCTION_BLOCK

{attribute 'OPC.UA.DA.JobMethod' := 'JobMethode_CompressorControl'}
FUNCTION_BLOCK MBS_VSG_AS_SuctionProcess
VAR
	AlwaysTrue : BOOL := TRUE;
	// Used for debugging purposes to display InputArguments of method call
	MethodCall_CompressorControl : BOOL := FALSE; // used to store InputArg "MethodCall" from Start() method
	ResetMethodCall	: BOOL := FALSE;
	Destination : STRING;
	callCounterStart : ULINT; // counts how many times the Start() method has been called
	callCounterCheckState : ULINT; // counts how many times the CheckState() method has been called
	callCounterAbort : ULINT; // counts how many times the Abort() method has been called
	
	// Variables to determine if a job has been started (Start() method has been called) or finished
	jobRunning : BOOL;
	jobFinished : BOOL;

	// State machine variable
	state : UDINT;
	
	//Variablen des Transport FBs
	MBS_VSG_SuctionProcess : CompressorControl;
END_VAR
	
VAR_INPUT
	ESS: BOOL;
	TouchSensor_01 : BOOL;
	TouchSensor_02 : BOOL;
	TON_PowerOnDelay_Compressor : TIME;
	TON_PowerOnDelay_Valve : TIME;
	AutomaticMode: BOOL;
END_VAR

VAR_OUTPUT
	DO_ControlCompressorSuctionProcessVSG_01 : BOOL;
	DO_ControlValveSuctionProcessVSG_02 : BOOL;
END_VAR

                  MBS_VSG_SuctionProcess(
    MethodCall := MethodCall_CompressorControl,
    EmergencyStopSignal := ESS,
    Destination := Destination,
    InitStateDrive_Input := ,
    DI01 := TouchSensor_01,
    DI02 := TouchSensor_02,
    DI03_EncoderStart01 := ,
    DI04_EncoderStart02 := ,
    DI05_EncoderStart03 := ,
    DI06_EncoderStart04 := ,
    DI07_EncoderStart05 := ,
    DI08_EncoderStart06 := ,
    DI09_EncoderTarget01 := ,
    DI10_EncoderTarget02 := ,
    DI11_EncoderTarget03 := ,
    DI12_EncoderTarget04 := ,
    DI13_EncoderTarget05 := ,
    DI14_EncoderTarget06 := ,
    PowerOFF_SelfSet := ,
    TON_Time_PowerOFFSelfSet := ,
    TON_Time_Compressor := TON_PowerOnDelay_Compressor,
    TON_Time_Valve := TON_PowerOnDelay_Valve,
    OperatingMode := AutomaticMode
);
DO_ControlCompressorSuctionProcessVSG_01 := MBS_VSG_SuctionProcess.DigitalOutputControl_01;
                

{attribute 'TcRpcEnable' := '1'}
METHOD Abort : HRESULT
VAR_INPUT
	hdl : UDINT; // Do not change, used by server.
END_VAR
                        callCounterAbort := callCounterAbort + 1;
                      
END_METHOD

{attribute 'TcRpcEnable' := '1'}
METHOD CheckState : HRESULT
VAR_INPUT
	hdl : UDINT; // Do not change, used by server.
END_VAR
VAR_OUTPUT
	bBusy : BOOL; // Do not change. Used by server to find out if the job is finished
	
	// List of OutputArguments for OPC UA method, may be customized
	State : BOOL; // Abgeschlossener MethodCall
	MethodCall: BOOL; //Input Recall
END_VAR
                        callCounterCheckState := callCounterCheckState + 1;
IF NOT jobFinished THEN
	bBusy := TRUE; // job is not finished yet
	CheckState := 0; // no error
ELSE
	bBusy := FALSE; // job is finished
	CheckState := 0; // done, no error occured during execution (OPC UA StatusCode "GOOD")
	jobFinished := FALSE;
	State := ResetMethodCall;
	MethodCall := MethodCall_CompressorControl;
END_IF
                      
END_METHOD

{attribute 'TcRpcEnable' := '1'}
METHOD Start : HRESULT
VAR_INPUT
	// List of InputArguments for OPC UA method, may be customized
	MethodCall : BOOL; // some description
	DestinationPoint : STRING;	
END_VAR
VAR_OUTPUT
	hdl : UDINT; // Do not change, used by server.
END_VAR
                        callCounterStart := callCounterStart + 1;

MethodCall_CompressorControl := MethodCall;
Destination := DestinationPoint;

jobRunning := TRUE;
Start := 0; // no error occured, e.g. while parsing the input arguments (0 = OPC UA StatusCode "GOOD")
                      
END_METHOD
END_FUNCTION_BLOCK

{attribute 'OPC.UA.DA.JobMethod' := 'JobMethode_CompressorControl'}
FUNCTION_BLOCK MBS_VSG_AS_VerticalMove
VAR
	AlwaysTrue : BOOL := TRUE;
	// Used for debugging purposes to display InputArguments of method call
	MethodCall_CompressorControl : BOOL := FALSE; // used to store InputArg "MethodCall" from Start() method
	ResetMethodCall	: BOOL := FALSE;
	DestinationVertical : STRING;
	PowerOFF_SelfSet : BOOL;
	PowerOFFDelay_SelfSet : TIME;
	callCounterStart : ULINT; // counts how many times the Start() method has been called
	callCounterCheckState : ULINT; // counts how many times the CheckState() method has been called
	callCounterAbort : ULINT; // counts how many times the Abort() method has been called
	
	// Variables to determine if a job has been started (Start() method has been called) or finished
	jobRunning : BOOL;
	jobFinished : BOOL;

	// State machine variable
	state : UDINT;
	
	//Variablen des Transport FBs
	MBS_VSG_VerticalMove : CompressorControl;
END_VAR
	
VAR_INPUT
	ESS: BOOL;
	TouchSensor_01 : BOOL;
	TON_PowerOnDelay_Compressor : TIME;
	TON_PowerOnDelay_Valve : TIME;
	AutomaticMode: BOOL;
END_VAR

VAR_OUTPUT
	DO_ControlCompressorVerticalMoveVSG_01 : BOOL;
	DO_ControlValveVerticalMoveVSG_02 : BOOL;
END_VAR

                  MBS_VSG_VerticalMove(
    MethodCall := MethodCall_CompressorControl,
    EmergencyStopSignal := ESS,
    Destination := DestinationVertical,
    InitStateDrive_Input := ,
    DI01 := TouchSensor_01,
    DI02 := ,
    DI03_EncoderStart01 := ,
    DI04_EncoderStart02 := ,
    DI05_EncoderStart03 := ,
    DI06_EncoderStart04 := ,
    DI07_EncoderStart05 := ,
    DI08_EncoderStart06 := ,
    DI09_EncoderTarget01 := ,
    DI10_EncoderTarget02 := ,
    DI11_EncoderTarget03 := ,
    DI12_EncoderTarget04 := ,
    DI13_EncoderTarget05 := ,
    DI14_EncoderTarget06 := ,
    PowerOFF_SelfSet := PowerOFF_SelfSet,
    TON_Time_PowerOFFSelfSet := PowerOFFDelay_SelfSet,
    TON_Time_Compressor := TON_PowerOnDelay_Compressor,
    TON_Time_Valve := TON_PowerOnDelay_Valve,
    OperatingMode := AutomaticMode
);
DO_ControlCompressorVerticalMoveVSG_01 := MBS_VSG_VerticalMove.DigitalOutputControl_01;

                

{attribute 'TcRpcEnable' := '1'}
METHOD Abort : HRESULT
VAR_INPUT
	hdl : UDINT; // Do not change, used by server.
END_VAR
                        callCounterAbort := callCounterAbort + 1;
                      
END_METHOD

{attribute 'TcRpcEnable' := '1'}
METHOD CheckState : HRESULT
VAR_INPUT
	hdl : UDINT; // Do not change, used by server.
END_VAR
VAR_OUTPUT
	bBusy : BOOL; // Do not change. Used by server to find out if the job is finished
	
	// List of OutputArguments for OPC UA method, may be customized
	State : BOOL; // Abgeschlossener MethodCall
	MethodCall: BOOL; //Input Recall
END_VAR
                        callCounterCheckState := callCounterCheckState + 1;
IF NOT jobFinished THEN
	bBusy := TRUE; // job is not finished yet
	CheckState := 0; // no error
ELSE
	bBusy := FALSE; // job is finished
	CheckState := 0; // done, no error occured during execution (OPC UA StatusCode "GOOD")
	jobFinished := FALSE;
	State := ResetMethodCall;
	MethodCall := MethodCall_CompressorControl;
END_IF
                      
END_METHOD

{attribute 'TcRpcEnable' := '1'}
METHOD Start : HRESULT
VAR_INPUT
	// List of InputArguments for OPC UA method, may be customized
	MethodCall : BOOL; // some description
	DestinationPoint : STRING;
	SelfSetPowerOff : BOOL;
	SelfSetPowerOffDelay : TIME;	
END_VAR
VAR_OUTPUT
	hdl : UDINT; // Do not change, used by server.
END_VAR
                        callCounterStart := callCounterStart + 1;

MethodCall_CompressorControl := MethodCall;
DestinationVertical := DestinationPoint;
PowerOFF_SelfSet := SelfSetPowerOff;
PowerOFFDelay_SelfSet := SelfSetPowerOffDelay;

jobRunning := TRUE;
Start := 0; // no error occured, e.g. while parsing the input arguments (0 = OPC UA StatusCode "GOOD")
                      
END_METHOD
END_FUNCTION_BLOCK

{attribute 'OPC.UA.DA.JobMethod' := 'JobMethode_HorizontalMove'}
FUNCTION_BLOCK SST_CB_AS_HorizontalMove
VAR
	AlwaysTrue : BOOL := TRUE;
	// Used for debugging purposes to display InputArguments of method call
	MethodCall_HorizontalMove : BOOL := FALSE; // used to store InputArg "MethodCall" from Start() method
	ResetMethodCall : BOOL := FALSE;	
	DirectionHorizontal : STRING;
//	TS_EndschalterEntlastung : BOOL;
	callCounterStart : ULINT; // counts how many times the Start() method has been called
	callCounterCheckState : ULINT; // counts how many times the CheckState() method has been called
	callCounterAbort : ULINT; // counts how many times the Abort() method has been called
	
	// Variables to determine if a job has been started (Start() method has been called) or finished
	jobRunning : BOOL;
	jobFinished : BOOL;

	// State machine variable
	state : UDINT;
	
	//Variablen des Transport FBs
	SST_CB_HorizontalMove : AxisControl_MultipleInputSensors;
END_VAR
	
VAR_INPUT
	ESS: BOOL;
	LightSensor_01 : BOOL;
	LightSensor_02 : BOOL;
	TOF_Time_Motoransteuerung : TIME;
	AutomaticMode : BOOL;
END_VAR

VAR_OUTPUT
	DO_MovingConveyorBelt : BOOL;
END_VAR

                  SST_CB_HorizontalMove(
    MethodCall := MethodCall_HorizontalMove,
    EmergencyStopSignal := ESS,
    Direction := DirectionHorizontal,
    InitStateDrive_Input := ,
    DI01 := LightSensor_01,
    DI02 := LightSensor_02,
    TouchSensorRelief := ,
    TOF_Time_MotorControl := TOF_Time_Motoransteuerung,
    TOF_Time_TouchSensorRelief := ,
    OperatingMode := AutomaticMode
);
DO_MovingConveyorBelt := SST_CB_HorizontalMove.DigitalOutputControl_01;
                

{attribute 'TcRpcEnable' := '1'}
METHOD Abort : HRESULT
VAR_INPUT
	hdl : UDINT; // Do not change, used by server.
END_VAR
                        callCounterAbort := callCounterAbort + 1;
                      
END_METHOD

{attribute 'TcRpcEnable' := '1'}
METHOD CheckState : HRESULT
VAR_INPUT
	hdl : UDINT; // Do not change, used by server.
END_VAR
VAR_OUTPUT
	bBusy : BOOL; // Do not change. Used by server to find out if the job is finished
	
	// List of OutputArguments for OPC UA method, may be customized
	State : BOOL; // Abgeschlossener MethodCall
	MethodCall: BOOL; //Input Recall
END_VAR
                        callCounterCheckState := callCounterCheckState + 1;
IF NOT jobFinished THEN
	bBusy := TRUE; // job is not finished yet
	CheckState := 0; // no error
ELSE
	bBusy := FALSE; // job is finished
	CheckState := 0; // done, no error occured during execution (OPC UA StatusCode "GOOD")
	jobFinished := FALSE;
	State := ResetMethodCall;
	MethodCall := MethodCall_HorizontalMove;
END_IF
                      
END_METHOD

{attribute 'TcRpcEnable' := '1'}
METHOD Start : HRESULT
VAR_INPUT
	// List of InputArguments for OPC UA method, may be customized
	MethodCall : BOOL; // some description
	DirectionPoint : STRING;
END_VAR
VAR_OUTPUT
	hdl : UDINT; // Do not change, used by server.
END_VAR
                        callCounterStart := callCounterStart + 1;

MethodCall_HorizontalMove := MethodCall;
DirectionHorizontal := DirectionPoint;

jobRunning := TRUE;
Start := 0; // no error occured, e.g. while parsing the input arguments (0 = OPC UA StatusCode "GOOD")
                      
END_METHOD
END_FUNCTION_BLOCK

{attribute 'OPC.UA.DA.JobMethod' := 'JobMethode_ColorDetection'}
FUNCTION_BLOCK SST_CS_AS_ColorDetection
VAR
	AlwaysTrue : BOOL := TRUE;
	// Used for debugging purposes to display InputArguments of method call
	MethodCall_ColorDetection : BOOL := FALSE; // used to store InputArg "MethodCall" from Start() method
	callCounterStart : ULINT; // counts how many times the Start() method has been called
	callCounterCheckState : ULINT; // counts how many times the CheckState() method has been called
	callCounterAbort : ULINT; // counts how many times the Abort() method has been called
	
	// Variables to determine if a job has been started (Start() method has been called) or finished
	jobRunning : BOOL;
	jobFinished : BOOL;

	// State machine variable
	state : UDINT;
	
	//Variablen des Transport FBs
	ResetCall : BOOL := FALSE;	
	SST_Auto_ColorDetection : AutomaticColorDetection_nichtfertig;
	
	//Farbcodes
	ColorCode1 : INT ;
	ColorCode2 : INT ;
	ColorCode3 : INT ;
END_VAR
	
VAR_INPUT
	Color_Sensor : INT;
END_VAR

VAR_OUTPUT
 Color_White : BOOL;
 Color_Red : BOOL;
 Color_Blue : BOOL;
END_VAR

                  SST_Auto_ColorDetection(ColorSensor := Color_Sensor, ColorCode_1 := ColorCode1, ColorCode_2 := ColorCode2, ColorCode_3 := ColorCode3);
Color_White := SST_Auto_ColorDetection.Color_1;
                

{attribute 'TcRpcEnable' := '1'}
METHOD Abort : HRESULT
VAR_INPUT
	hdl : UDINT; // Do not change, used by server.
END_VAR
                        callCounterAbort := callCounterAbort + 1;
                      
END_METHOD

{attribute 'TcRpcEnable' := '1'}
METHOD CheckState : HRESULT
VAR_INPUT
	hdl : UDINT; // Do not change, used by server.
END_VAR
VAR_OUTPUT
	bBusy : BOOL; // Do not change. Used by server to find out if the job is finished
	
	// List of OutputArguments for OPC UA method, may be customized
	State : BOOL; // Abgeschlossener MethodCall
	MethodCall: BOOL; //Input Recall
END_VAR
                        callCounterCheckState := callCounterCheckState + 1;
IF NOT jobFinished THEN
	bBusy := TRUE; // job is not finished yet
	CheckState := 0; // no error
ELSE
	bBusy := FALSE; // job is finished
	CheckState := 0; // done, no error occured during execution (OPC UA StatusCode "GOOD")
	jobFinished := FALSE;
	State := ResetCall;
	MethodCall := MethodCall_ColorDetection;
END_IF
                      
END_METHOD

{attribute 'TcRpcEnable' := '1'}
METHOD Start : HRESULT
VAR_INPUT
	// List of InputArguments for OPC UA method, may be customized
	MethodCall : BOOL; // some description
	DirectionPointA : BOOL;
	DirectionPointB : BOOL;
	EndschalterEntlastung : BOOL;	
END_VAR
VAR_OUTPUT
	hdl : UDINT; // Do not change, used by server.
END_VAR
                        callCounterStart := callCounterStart + 1;

MethodCall_ColorDetection := MethodCall;

jobRunning := TRUE;
Start := 0; // no error occured, e.g. while parsing the input arguments (0 = OPC UA StatusCode "GOOD")
                      
END_METHOD
END_FUNCTION_BLOCK

{attribute 'OPC.UA.DA.JobMethod' := 'JobMethode_CompressorControl'}
FUNCTION_BLOCK SST_PD_AS_HorizontalMove
VAR
	AlwaysTrue : BOOL := TRUE;
	// Used for debugging purposes to display InputArguments of method call
	MethodCall_CompressorControl : BOOL := FALSE; // used to store InputArg "MethodCall" from Start() method
	ResetMethodCall : BOOL := FALSE;
	DestinationHorizontal : STRING;
	callCounterStart : ULINT; // counts how many times the Start() method has been called
	callCounterCheckState : ULINT; // counts how many times the CheckState() method has been called
	callCounterAbort : ULINT; // counts how many times the Abort() method has been called
	
	// Variables to determine if a job has been started (Start() method has been called) or finished
	jobRunning : BOOL;
	jobFinished : BOOL;

	// State machine variable
	state : UDINT;
	
	//Variablen des Transport FBs
	
	MBS_VSG_HorizontalMove : CompressorControl;
END_VAR
	
VAR_INPUT
	ESS: BOOL;
	LightSensor_01 : BOOL;
	LightSensor_02 : BOOL;
	PowerOnDelay_Compressor : TIME;
	PowerOnDelay_Valve : TIME;
	AutomaticMode : BOOL;
END_VAR

VAR_OUTPUT
	DO_ControlCompressorPD_01 : BOOL;
	DO_ControlValvePD_02 : BOOL;
END_VAR

                  MBS_VSG_HorizontalMove(
    MethodCall := MethodCall_CompressorControl,
    EmergencyStopSignal := ESS,
    Destination := DestinationHorizontal,
    InitStateDrive_Input := ,
    DI01 := LightSensor_01,
    DI02 := LightSensor_02,
    DI03_EncoderStart01 := ,
    DI04_EncoderStart02 := ,
    DI05_EncoderStart03 := ,
    DI06_EncoderStart04 := ,
    DI07_EncoderStart05 := ,
    DI08_EncoderStart06 := ,
    DI09_EncoderTarget01 := ,
    DI10_EncoderTarget02 := ,
    DI11_EncoderTarget03 := ,
    DI12_EncoderTarget04 := ,
    DI13_EncoderTarget05 := ,
    DI14_EncoderTarget06 := ,
    PowerOFF_SelfSet := ,
    TON_Time_PowerOFFSelfSet := ,
    TON_Time_Compressor := PowerOnDelay_Compressor,
    TON_Time_Valve := PowerOnDelay_Valve,
    OperatingMode := AutomaticMode
);
DO_ControlCompressorPD_01 := MBS_VSG_HorizontalMove.DigitalOutputControl_01;
                

{attribute 'TcRpcEnable' := '1'}
METHOD Abort : HRESULT
VAR_INPUT
	hdl : UDINT; // Do not change, used by server.
END_VAR
                        callCounterAbort := callCounterAbort + 1;
                      
END_METHOD

{attribute 'TcRpcEnable' := '1'}
METHOD CheckState : HRESULT
VAR_INPUT
	hdl : UDINT; // Do not change, used by server.
END_VAR
VAR_OUTPUT
	bBusy : BOOL; // Do not change. Used by server to find out if the job is finished
	
	// List of OutputArguments for OPC UA method, may be customized
	State : BOOL; // Abgeschlossener MethodCall
	MethodCall: BOOL; //Input Recall
END_VAR
                        callCounterCheckState := callCounterCheckState + 1;
IF NOT jobFinished THEN
	bBusy := TRUE; // job is not finished yet
	CheckState := 0; // no error
ELSE
	bBusy := FALSE; // job is finished
	CheckState := 0; // done, no error occured during execution (OPC UA StatusCode "GOOD")
	jobFinished := FALSE;
	State := ResetMethodCall;
	MethodCall := MethodCall_CompressorControl;
END_IF
                      
END_METHOD

{attribute 'TcRpcEnable' := '1'}
METHOD Start : HRESULT
VAR_INPUT
	// List of InputArguments for OPC UA method, may be customized
	MethodCall : BOOL; // some description
	DestinationPoint : STRING;	
END_VAR
VAR_OUTPUT
	hdl : UDINT; // Do not change, used by server.
END_VAR
                        callCounterStart := callCounterStart + 1;

MethodCall_CompressorControl := MethodCall;
DestinationHorizontal := DestinationPoint;

jobRunning := TRUE;
Start := 0; // no error occured, e.g. while parsing the input arguments (0 = OPC UA StatusCode "GOOD")
                      
END_METHOD
END_FUNCTION_BLOCK

{attribute 'OPC.UA.DA.JobMethod' := 'JobMethode_CompressorControl'}
FUNCTION_BLOCK VSG_AS_CompressorControl
VAR
    MethodCall_CompressorControl : BOOL := FALSE;
    ResetMethodCall : BOOL := FALSE;

    Destination : BOOL := TRUE;

    EncoderTargetPosition01 : UDINT;
    EncoderTargetPosition02 : UDINT;
    EncoderTargetPosition03 : UDINT;
    EncoderTargetPosition04 : UDINT;
    EncoderTargetPosition05 : UDINT;
    EncoderTargetPosition06 : UDINT;

    callCounterStart : ULINT;
    callCounterCheckState : ULINT;
    callCounterAbort : ULINT;

    jobRunning : BOOL := FALSE;
    jobFinished : BOOL := FALSE;
    state : UDINT := 0;

    MBS_VSG_VerticalMove : CompressorControl;

    TON_TimeCompressor : TIME := T#0MS;
    TON_TimeValve : TIME := T#0MS;
    TON_TimePowerOffSelfSet : TIME := T#100MS;

    PowerOffSelfSet : BOOL := TRUE;
END_VAR

VAR_INPUT
    ESS : BOOL;

    EncoderStartPosition01 : UDINT;
    EncoderStartPosition02 : UDINT;
    EncoderStartPosition03 : UDINT;
    EncoderStartPosition04 : UDINT;
    EncoderStartPosition05 : UDINT;
    EncoderStartPosition06 : UDINT;

    WorkpieceAtPickupPosition : BOOL;
    AutomaticMode : BOOL;
END_VAR

VAR_OUTPUT
    DO_CompressorVSG : BOOL;
    DO_ValveVSG : BOOL;

    VSG_ErrorDetected : BOOL;
    VSG_ErrorCode : UDINT;
END_VAR

                  //VSG_ErrorDetected := FALSE;
//VSG_ErrorCode := 0;

IF MethodCall_CompressorControl AND NOT WorkpieceAtPickupPosition THEN

    VSG_ErrorDetected := TRUE;
    VSG_ErrorCode := 1001;

    DO_CompressorVSG := FALSE;
    DO_ValveVSG := FALSE;

    MethodCall_CompressorControl := FALSE;
    ResetMethodCall := TRUE;

    jobRunning := FALSE;
    jobFinished := TRUE;
    state := 900;

ELSE

    MBS_VSG_VerticalMove(
        MethodCall := MethodCall_CompressorControl,
        EmergencyStopSignal := NOT ESS,
        Destination := Destination,
        InitStateDrive_Input := FALSE,

        DI01 := WorkpieceAtPickupPosition,
        DI02 := FALSE,

        DI03_EncoderStart01 := EncoderStartPosition01,
        DI04_EncoderStart02 := EncoderStartPosition02,
        DI05_EncoderStart03 := EncoderStartPosition03,
        DI06_EncoderStart04 := EncoderStartPosition04,
        DI07_EncoderStart05 := EncoderStartPosition05,
        DI08_EncoderStart06 := EncoderStartPosition06,

        DI09_EncoderTarget01 := EncoderTargetPosition01,
        DI10_EncoderTarget02 := EncoderTargetPosition02,
        DI11_EncoderTarget03 := EncoderTargetPosition03,
        DI12_EncoderTarget04 := EncoderTargetPosition04,
        DI13_EncoderTarget05 := EncoderTargetPosition05,
        DI14_EncoderTarget06 := EncoderTargetPosition06,

        PowerOFF_SelfSet := PowerOffSelfSet,
        TON_Time_PowerOFFSelfSet := TON_TimePowerOffSelfSet,
        TON_Time_Compressor := TON_TimeCompressor,
        TON_Time_Valve := TON_TimeValve,
        OperatingMode := AutomaticMode
    );

    DO_CompressorVSG := MBS_VSG_VerticalMove.DigitalOutputControl_01;
    DO_ValveVSG := MBS_VSG_VerticalMove.DigitalOutputControl_02;
    ResetMethodCall := MBS_VSG_VerticalMove.ResetMethodCall;

    IF ResetMethodCall THEN
        MethodCall_CompressorControl := FALSE;
        jobRunning := FALSE;
        jobFinished := TRUE;
        state := 100;
    END_IF;

END_IF;
                

{attribute 'TcRpcEnable' := '1'}
METHOD Abort : HRESULT
VAR_INPUT
    hdl : UDINT;
END_VAR
                        callCounterAbort := callCounterAbort + 1;

MethodCall_CompressorControl := FALSE;
ResetMethodCall := TRUE;

DO_CompressorVSG := FALSE;
DO_ValveVSG := FALSE;

jobRunning := FALSE;
jobFinished := TRUE;
state := 999;

Abort := 0;
                      
END_METHOD

{attribute 'TcRpcEnable' := '1'}
METHOD CheckState : HRESULT
VAR_INPUT
    hdl : UDINT;
END_VAR

VAR_OUTPUT
    bBusy : BOOL;
    State : UDINT;
    IsDone : BOOL;
    HasError : BOOL;
    ErrorCode : UDINT;
END_VAR
                        callCounterCheckState := callCounterCheckState + 1;

bBusy := jobRunning;
State := state;
IsDone := jobFinished;
HasError := VSG_ErrorDetected;
ErrorCode := VSG_ErrorCode;

CheckState := 0;
                      
END_METHOD

{attribute 'TcRpcEnable' := '1'}
METHOD Start : HRESULT
VAR_INPUT
    MethodCall : BOOL;
    DestinationReached : BOOL;
    EncoderTargetPosition_01 : UDINT;
    EncoderTargetPosition_02 : UDINT;
    EncoderTargetPosition_03 : UDINT;
    EncoderTargetPosition_04 : UDINT;
    EncoderTargetPosition_05 : UDINT;
    EncoderTargetPosition_06 : UDINT;
END_VAR

VAR_OUTPUT
    hdl : UDINT;
END_VAR
                        callCounterStart := callCounterStart + 1;

IF NOT jobRunning THEN
	
	IF MethodCall THEN
        OPCUA.lastExecutedProcess := 'VSG_Skill_SuctionProcess';
        OPCUA.lastExecutedSkill := 'VSG_AS_CompressorControl';
    END_IF;
	
    MethodCall_CompressorControl := MethodCall;
    Destination := DestinationReached;

    EncoderTargetPosition01 := EncoderTargetPosition_01;
    EncoderTargetPosition02 := EncoderTargetPosition_02;
    EncoderTargetPosition03 := EncoderTargetPosition_03;
    EncoderTargetPosition04 := EncoderTargetPosition_04;
    EncoderTargetPosition05 := EncoderTargetPosition_05;
    EncoderTargetPosition06 := EncoderTargetPosition_06;

    jobRunning := TRUE;
    jobFinished := FALSE;
    state := 1;

    hdl := 1;
    Start := 0;

ELSE

    hdl := 0;
    Start := 16#800700AA;

END_IF;
                      
END_METHOD
END_FUNCTION_BLOCK

{attribute 'OPC.UA.DA.JobMethod' := 'JobMethode_HorizontalMove'}
FUNCTION_BLOCK VSG_AS_HorizontalMoveEncoder
VAR
    MethodCall_HorizontalMove : BOOL := FALSE;
    ResetMethodCall : BOOL := FALSE;

    DirectionHorizontal : BOOL := TRUE;

    EncoderTargetPosition01 : UDINT;
    EncoderTargetPosition02 : UDINT;

    TSR : BOOL := FALSE;

    callCounterStart : ULINT;
    callCounterCheckState : ULINT;
    callCounterAbort : ULINT;

    jobRunning : BOOL := FALSE;
    jobFinished : BOOL := FALSE;
    state : UDINT := 0;

    VSG_HorizontalMoveWithEncoder : AxisControl_Encoder;
END_VAR

VAR_INPUT
    ESS : BOOL;
    TouchSensor01 : BOOL;
    EncoderStartPosition01 : UDINT;
    EncoderStartPosition02 : UDINT;
    TOF_Time_TSR : TIME;
    AutomaticMode : BOOL;
END_VAR

VAR_OUTPUT
    DO_MovingHorizontalVSG_01 : BOOL;
END_VAR

                  VSG_HorizontalMoveWithEncoder(
    MethodCall := MethodCall_HorizontalMove,
    EmergencyStopSignal := NOT ESS,
    Direction := DirectionHorizontal,
    InitStateDrive_Input := FALSE,
    DI01 := TouchSensor01,
    DI02_EncoderStart01 := EncoderStartPosition01,
    DI03_EncoderTarget01 := EncoderTargetPosition01,
    DI04_EncoderStart02 := EncoderStartPosition02,
    DI05_EncoderTarget02 := EncoderTargetPosition02,
    TouchSensorRelief := TSR,
    TOF_Time_MotorControl := T#0MS,
    TOF_Time_TouchSensorRelief := TOF_Time_TSR,
    OperatingMode := AutomaticMode
);

DO_MovingHorizontalVSG_01 := VSG_HorizontalMoveWithEncoder.DigitalOutputControl_01;
ResetMethodCall := VSG_HorizontalMoveWithEncoder.ResetMethodCall;

IF ResetMethodCall THEN
    MethodCall_HorizontalMove := FALSE;
    jobRunning := FALSE;
    jobFinished := TRUE;
    state := 100;
END_IF;
                

{attribute 'TcRpcEnable' := '1'}
METHOD Abort : HRESULT
VAR_INPUT
    hdl : UDINT;
END_VAR
                        callCounterAbort := callCounterAbort + 1;

MethodCall_HorizontalMove := FALSE;
DO_MovingHorizontalVSG_01 := FALSE;

jobRunning := FALSE;
jobFinished := TRUE;
state := 999;

Abort := 0;
                      
END_METHOD

{attribute 'TcRpcEnable' := '1'}
METHOD CheckState : HRESULT
VAR_INPUT
    hdl : UDINT;
END_VAR

VAR_OUTPUT
    bBusy : BOOL;
    State : UDINT;
    IsDone : BOOL;
END_VAR
                        callCounterCheckState := callCounterCheckState + 1;

bBusy := jobRunning;
State := state;
IsDone := jobFinished;

CheckState := 0;
                      
END_METHOD

{attribute 'TcRpcEnable' := '1'}
METHOD Start : HRESULT
VAR_INPUT
    MethodCall : BOOL;
    MovementDirection : BOOL;
    EncoderPositionHorizontal_01 : UDINT;
    EncoderPositionHorizontal_02 : UDINT;
    TouchSensorRelief : BOOL;
END_VAR

VAR_OUTPUT
    hdl : UDINT;
END_VAR
                        callCounterStart := callCounterStart + 1;

IF NOT jobRunning THEN

    MethodCall_HorizontalMove := MethodCall;
    DirectionHorizontal := MovementDirection;

    EncoderTargetPosition01 := EncoderPositionHorizontal_01;
    EncoderTargetPosition02 := EncoderPositionHorizontal_02;

    TSR := TouchSensorRelief;

    jobRunning := TRUE;
    jobFinished := FALSE;
    state := 1;

    hdl := 1;
    Start := 0;

ELSE

    hdl := 0;
    Start := 16#800700AA;

END_IF;
                      
END_METHOD
END_FUNCTION_BLOCK

{attribute 'OPC.UA.DA.JobMethod' := 'JobMethode_RotationMove'}
FUNCTION_BLOCK VSG_AS_RotationMoveEncoder
VAR
    MethodCall_RotationMove : BOOL := FALSE;
    ResetMethodCall : BOOL := FALSE;

    DirectionRotation : BOOL := TRUE;

    EncoderTargetPosition01 : UDINT;
    EncoderTargetPosition02 : UDINT;

    TSR : BOOL := FALSE;

    callCounterStart : ULINT;
    callCounterCheckState : ULINT;
    callCounterAbort : ULINT;

    jobRunning : BOOL := FALSE;
    jobFinished : BOOL := FALSE;
    state : UDINT := 0;

    VSG_RotationMoveWithEncoder : AxisControl_Encoder;
END_VAR

VAR_INPUT
    ESS : BOOL;
    TouchSensor01 : BOOL;
    EncoderStartPosition01 : UDINT;
    EncoderStartPosition02 : UDINT;
    TOF_Time_TSR : TIME;
    AutomaticMode : BOOL;
END_VAR

VAR_OUTPUT
    DO_MovingRotationVSG_01 : BOOL;
END_VAR

                  VSG_RotationMoveWithEncoder(
    MethodCall := MethodCall_RotationMove,
    EmergencyStopSignal := NOT ESS,
    Direction := DirectionRotation,
    InitStateDrive_Input := FALSE,
    DI01 := TouchSensor01,
    DI02_EncoderStart01 := EncoderStartPosition01,
    DI03_EncoderTarget01 := EncoderTargetPosition01,
    DI04_EncoderStart02 := EncoderStartPosition02,
    DI05_EncoderTarget02 := EncoderTargetPosition02,
    TouchSensorRelief := TSR,
    TOF_Time_MotorControl := T#0MS,
    TOF_Time_TouchSensorRelief := TOF_Time_TSR,
    OperatingMode := AutomaticMode
);

DO_MovingRotationVSG_01 := VSG_RotationMoveWithEncoder.DigitalOutputControl_01;
ResetMethodCall := VSG_RotationMoveWithEncoder.ResetMethodCall;

